LIN {X 0,Y 467.531,Z 199.445,A -85,B 0,C 180,E1 -7625.111,E2 -7625.111} C_VEL
LIN {X 0,Y 467.326,Z 207.202,A -85,B 0,C 180,E1 -7628.383,E2 -7628.383} C_VEL
LIN {X 0,Y 467.095,Z 214.915,A -85,B 0,C 180,E1 -7631.583,E2 -7631.583} C_VEL
LIN {X 0,Y 466.901,Z 222.309,A -85,B 0,C 180,E1 -7634.625,E2 -7634.625} C_VEL
LIN {X 0,Y 469.16,Z 236.323,A -85,B 0,C 180,E1 -7635.082,E2 -7635.082} C_VEL
LIN {X 0,Y 469.908,Z 243.542,A -85,B 0,C 180,E1 -7635.383,E2 -7635.383} C_VEL
LIN {X 0,Y 469.499,Z 254.745,A -85,B 0,C 180,E1 -7635.923,E2 -7635.923} C_VEL
LIN {X 0,Y 468.983,Z 266.744,A -85,B 0,C 180,E1 -7636.681,E2 -7636.681} C_VEL
LIN {X 0,Y 468.599,Z 277.34,A -85,B 0,C 180,E1 -7637.54,E2 -7637.54} C_VEL
LIN {X 0,Y 468.086,Z 287.224,A -85,B 0,C 180,E1 -7638.526,E2 -7638.526} C_VEL
LIN {X 0,Y 467.594,Z 296.115,A -85,B 0,C 180,E1 -7639.611,E2 -7639.611} C_VEL
LIN {X 0,Y 467.253,Z 304.795,A -85,B 0,C 180,E1 -7640.914,E2 -7640.914} C_VEL
LIN {X 0,Y 466.98,Z 311.72,A -85,B 0,C 180,E1 -7642.217,E2 -7642.217} C_VEL
LIN {X 0,Y 466.805,Z 317.387,A -85,B 0,C 180,E1 -7643.549,E2 -7643.549} C_VEL
LIN {X 0,Y 466.739,Z 321.625,A -85,B 0,C 180,E1 -7644.817,E2 -7644.817} C_VEL
LIN {X 0,Y 466.646,Z 323.927,A -85,B 0,C 180,E1 -7645.682,E2 -7645.682} C_VEL
LIN {X 0,Y 466.688,Z 325.799,A -85,B 0,C 180,E1 -7646.547,E2 -7646.547} C_VEL
LIN {X 0,Y 466.662,Z 327.203,A -85,B 0,C 180,E1 -7647.411,E2 -7647.411} C_VEL
LIN {X 0,Y 466.618,Z 328.815,A -85,B 0,C 180,E1 -7649.138,E2 -7649.138} C_VEL
LIN {X 0,Y 466.599,Z 329.038,A -85,B 0,C 180,E1 -7650.001,E2 -7650.001} C_VEL
LIN {X 0,Y 466.618,Z 328.829,A -85,B 0,C 180,E1 -7650.864,E2 -7650.864} C_VEL
LIN {X 0,Y 466.662,Z 327.238,A -85,B 0,C 180,E1 -7652.59,E2 -7652.59} C_VEL
LIN {X 0,Y 466.688,Z 325.85,A -85,B 0,C 180,E1 -7653.454,E2 -7653.454} C_VEL
LIN {X 0,Y 466.689,Z 322.925,A -85,B 0,C 180,E1 -7654.751,E2 -7654.751} C_VEL
LIN {X 0,Y 466.753,Z 318.967,A -85,B 0,C 180,E1 -7656.05,E2 -7656.05} C_VEL
LIN {X 0,Y 466.963,Z 312.888,A -85,B 0,C 180,E1 -7657.567,E2 -7657.567} C_VEL
LIN {X 0,Y 467.224,Z 306.239,A -85,B 0,C 180,E1 -7658.869,E2 -7658.869} C_VEL
LIN {X 0,Y 467.551,Z 297.991,A -85,B 0,C 180,E1 -7660.173,E2 -7660.173} C_VEL
LIN {X 0,Y 468.052,Z 289.556,A -85,B 0,C 180,E1 -7661.256,E2 -7661.256} C_VEL
LIN {X 0,Y 468.503,Z 279.581,A -85,B 0,C 180,E1 -7662.301,E2 -7662.301} C_VEL
LIN {X 0,Y 468.948,Z 268.843,A -85,B 0,C 180,E1 -7663.211,E2 -7663.211} C_VEL
LIN {X 0,Y 469.452,Z 257.578,A -85,B 0,C 180,E1 -7663.969,E2 -7663.969} C_VEL
LIN {X 0,Y 469.965,Z 246.132,A -85,B 0,C 180,E1 -7664.561,E2 -7664.561} C_VEL
LIN {X 0,Y 469.806,Z 241.144,A -85,B 0,C 180,E1 -7664.78,E2 -7664.78} C_VEL
LIN {X 0,Y 468.016,Z 228.536,A -85,B 0,C 180,E1 -7665.256,E2 -7665.256} C_VEL
LIN {X 0,Y 466.938,Z 222.233,A -85,B 0,C 180,E1 -7665.454,E2 -7665.454} C_VEL
LIN {X 0,Y 467.097,Z 214.666,A -85,B 0,C 180,E1 -7668.575,E2 -7668.575} C_VEL
LIN {X 0,Y 467.326,Z 207.444,A -85,B 0,C 180,E1 -7671.619,E2 -7671.619} C_VEL
LIN {X 0,Y 467.555,Z 199.754,A -85,B 0,C 180,E1 -7674.889,E2 -7674.889} C_VEL
LIN {X 0,Y 467.862,Z 192.074,A -85,B 0,C 180,E1 -7678.239,E2 -7678.239} C_VEL
LIN {X 0,Y 468.123,Z 186.635,A -85,B 0,C 180,E1 -7680.692,E2 -7680.692} C_VEL
LIN {X 0,Y 468.345,Z 182.022,A -85,B 0,C 180,E1 -7682.824,E2 -7682.824} C_VEL
LIN {X 0,Y 468.553,Z 176.91,A -85,B 0,C 180,E1 -7685.271,E2 -7685.271} C_VEL
LIN {X 0,Y 468.198,Z 172.916,A -85,B 0,C 180,E1 -7687.291,E2 -7687.291} C_VEL
LIN {X 0,Y 467.587,Z 169.247,A -85,B 0,C 180,E1 -7689.28,E2 -7689.28} C_VEL
LIN {X 0,Y 467.608,Z 169.237,A -85,B 0,C 180,E1 -7692.57,E2 -7692.57} C_VEL
LIN {X 0,Y 467.557,Z 169.245,A -85,B 0,C 180,E1 -7695.051,E2 -7695.051} C_VEL
LIN {X 0,Y 467.575,Z 169.243,A -85,B 0,C 180,E1 -7697.438,E2 -7697.438} C_VEL
LIN {X 0,Y 467.543,Z 169.247,A -85,B 0,C 180,E1 -7700.851,E2 -7700.851} C_VEL
LIN {X 0,Y 467.545,Z 169.243,A -85,B 0,C 180,E1 -7704.259,E2 -7704.259} C_VEL
LIN {X 0,Y 467.562,Z 169.245,A -85,B 0,C 180,E1 -7707.319,E2 -7707.319} C_VEL
LIN {X 0,Y 467.549,Z 169.247,A -85,B 0,C 180,E1 -7710.666,E2 -7710.666} C_VEL
LIN {X 0,Y 467.594,Z 169.241,A -85,B 0,C 180,E1 -7713.198,E2 -7713.198} C_VEL
LIN {X 0,Y 467.584,Z 169.24,A -85,B 0,C 180,E1 -7716.463,E2 -7716.463} C_VEL
LIN {X 0,Y 467.601,Z 169.237,A -85,B 0,C 180,E1 -7719.776,E2 -7719.776} C_VEL
LIN {X 0,Y 467.594,Z 169.242,A -85,B 0,C 180,E1 -7722.506,E2 -7722.506} C_VEL
LIN {X 0,Y 467.578,Z 169.243,A -85,B 0,C 180,E1 -7725.196,E2 -7725.196} C_VEL
LIN {X 0,Y 467.658,Z 169.231,A -85,B 0,C 180,E1 -7727.855,E2 -7727.855} C_VEL
LIN {X 0,Y 467.671,Z 169.227,A -85,B 0,C 180,E1 -7731.357,E2 -7731.357} C_VEL
LIN {X 0,Y 467.745,Z 169.222,A -85,B 0,C 180,E1 -7733.963,E2 -7733.963} C_VEL
LIN {X 0,Y 467.831,Z 169.21,A -85,B 0,C 180,E1 -7737.417,E2 -7737.417} C_VEL
LIN {X 0,Y 467.8,Z 169.213,A -85,B 0,C 180,E1 -7740.861,E2 -7740.861} C_VEL
LIN {X 0,Y 467.842,Z 169.208,A -85,B 0,C 180,E1 -7742.583,E2 -7742.583} C_VEL
LIN {X 0,Y 467.728,Z 169.225,A -85,B 0,C 180,E1 -7746.038,E2 -7746.038} C_VEL
LIN {X 0,Y 467.655,Z 169.232,A -85,B 0,C 180,E1 -7748.644,E2 -7748.644} C_VEL
LIN {X 0,Y 467.629,Z 169.238,A -85,B 0,C 180,E1 -7752.146,E2 -7752.146} C_VEL
LIN {X 0,Y 467.642,Z 169.235,A -85,B 0,C 180,E1 -7755.894,E2 -7755.894} C_VEL
LIN {X 0,Y 467.602,Z 169.241,A -85,B 0,C 180,E1 -7759.309,E2 -7759.309} C_VEL
LIN {X 0,Y 467.517,Z 169.25,A -85,B 0,C 180,E1 -7762.075,E2 -7762.075} C_VEL
LIN {X 0,Y 467.581,Z 169.241,A -85,B 0,C 180,E1 -7764.889,E2 -7764.889} C_VEL
LIN {X 0,Y 467.601,Z 169.239,A -85,B 0,C 180,E1 -7767.771,E2 -7767.771} C_VEL
LIN {X 0,Y 467.553,Z 169.248,A -85,B 0,C 180,E1 -7771.047,E2 -7771.047} C_VEL
LIN {X 0,Y 467.572,Z 169.242,A -85,B 0,C 180,E1 -7774.244,E2 -7774.244} C_VEL
LIN {X 0,Y 467.532,Z 169.249,A -85,B 0,C 180,E1 -7777.188,E2 -7777.188} C_VEL
LIN {X 0,Y 467.56,Z 169.242,A -85,B 0,C 180,E1 -7780.267,E2 -7780.267} C_VEL
LIN {X 0,Y 467.574,Z 169.243,A -85,B 0,C 180,E1 -7782.569,E2 -7782.569} C_VEL
LIN {X 0,Y 467.559,Z 169.244,A -85,B 0,C 180,E1 -7785.055,E2 -7785.055} C_VEL
LIN {X 0,Y 467.58,Z 169.241,A -85,B 0,C 180,E1 -7787.442,E2 -7787.442} C_VEL
LIN {X 0,Y 467.563,Z 169.244,A -85,B 0,C 180,E1 -7790.049,E2 -7790.049} C_VEL
LIN {X 0,Y 467.489,Z 169.254,A -85,B 0,C 180,E1 -7791.951,E2 -7791.951} C_VEL
LIN {X 0,Y 467.443,Z 170.109,A -85,B 0,C 180,E1 -7793.032,E2 -7793.032} C_VEL
LIN {X 0,Y 467.424,Z 173.846,A -85,B 0,C 180,E1 -7795.788,E2 -7795.788} C_VEL
LIN {X 0,Y 467.292,Z 178.365,A -85,B 0,C 180,E1 -7799.012,E2 -7799.012} C_VEL
LIN {X 0,Y 467.153,Z 182.951,A -85,B 0,C 180,E1 -7802.202,E2 -7802.202} C_VEL
LIN {X 0,Y 467.065,Z 187.177,A -85,B 0,C 180,E1 -7805.083,E2 -7805.083} C_VEL
LIN {X 0,Y 466.926,Z 191.458,A -85,B 0,C 180,E1 -7807.897,E2 -7807.897} C_VEL
LIN {X 0,Y 466.869,Z 196.787,A -85,B 0,C 180,E1 -7811.32,E2 -7811.32} C_VEL
LIN {X 0,Y 466.799,Z 198.848,A -85,B 0,C 180,E1 -7812.63,E2 -7812.63} C_VEL
LIN {X 0,Y 469.626,Z 212.179,A -85,B 0,C 180,E1 -7813.118,E2 -7813.118} C_VEL
LIN {X 0,Y 470.304,Z 216.846,A -85,B 0,C 180,E1 -7813.322,E2 -7813.322} C_VEL
LIN {X 0,Y 470.182,Z 221.204,A -85,B 0,C 180,E1 -7813.507,E2 -7813.507} C_VEL
LIN {X 0,Y 469.309,Z 226.817,A -85,B 0,C 180,E1 -7813.759,E2 -7813.759} C_VEL
LIN {X 0,Y 464.784,Z 238.986,A -85,B 0,C 180,E1 -7814.361,E2 -7814.361} C_VEL
LIN {X 0,Y 462.582,Z 245.641,A -85,B 0,C 180,E1 -7814.797,E2 -7814.797} C_VEL
LIN {X 0,Y 462.098,Z 248.855,A -85,B 0,C 180,E1 -7815.056,E2 -7815.056} C_VEL
LIN {X 0,Y 461.556,Z 259.922,A -85,B 0,C 180,E1 -7816.124,E2 -7816.124} C_VEL
LIN {X 0,Y 461.031,Z 269.785,A -85,B 0,C 180,E1 -7817.325,E2 -7817.325} C_VEL
LIN {X 0,Y 460.671,Z 278.005,A -85,B 0,C 180,E1 -7818.561,E2 -7818.561} C_VEL
LIN {X 0,Y 460.209,Z 285.169,A -85,B 0,C 180,E1 -7819.885,E2 -7819.885} C_VEL
LIN {X 0,Y 459.987,Z 290.869,A -85,B 0,C 180,E1 -7821.212,E2 -7821.212} C_VEL
LIN {X 0,Y 459.795,Z 295.352,A -85,B 0,C 180,E1 -7822.535,E2 -7822.535} C_VEL
LIN {X 0,Y 459.673,Z 298.757,A -85,B 0,C 180,E1 -7823.856,E2 -7823.856} C_VEL
LIN {X 0,Y 459.645,Z 300.447,A -85,B 0,C 180,E1 -7824.736,E2 -7824.736} C_VEL
LIN {X 0,Y 459.613,Z 302.633,A -85,B 0,C 180,E1 -7826.493,E2 -7826.493} C_VEL
LIN {X 0,Y 459.585,Z 303.127,A -85,B 0,C 180,E1 -7827.37,E2 -7827.37} C_VEL
LIN {X 0,Y 459.525,Z 302.9,A -85,B 0,C 180,E1 -7829.123,E2 -7829.123} C_VEL
LIN {X 0,Y 459.535,Z 302.217,A -85,B 0,C 180,E1 -7829.999,E2 -7829.999} C_VEL
LIN {X 0,Y 459.562,Z 301.135,A -85,B 0,C 180,E1 -7830.876,E2 -7830.876} C_VEL
LIN {X 0,Y 459.629,Z 299.611,A -85,B 0,C 180,E1 -7831.752,E2 -7831.752} C_VEL
LIN {X 0,Y 459.785,Z 296.553,A -85,B 0,C 180,E1 -7833.066,E2 -7833.066} C_VEL
LIN {X 0,Y 459.934,Z 292.454,A -85,B 0,C 180,E1 -7834.381,E2 -7834.381} C_VEL
LIN {X 0,Y 460.123,Z 286.196,A -85,B 0,C 180,E1 -7835.917,E2 -7835.917} C_VEL
LIN {X 0,Y 460.556,Z 278.996,A -85,B 0,C 180,E1 -7837.299,E2 -7837.299} C_VEL
LIN {X 0,Y 460.913,Z 270.853,A -85,B 0,C 180,E1 -7838.549,E2 -7838.549} C_VEL
LIN {X 0,Y 461.396,Z 262.105,A -85,B 0,C 180,E1 -7839.644,E2 -7839.644} C_VEL
LIN {X 0,Y 461.917,Z 251.339,A -85,B 0,C 180,E1 -7840.74,E2 -7840.74} C_VEL
LIN {X 0,Y 462.429,Z 240.492,A -85,B 0,C 180,E1 -7841.616,E2 -7841.616} C_VEL
LIN {X 0,Y 462.913,Z 228.195,A -85,B 0,C 180,E1 -7842.39,E2 -7842.39} C_VEL
LIN {X 0,Y 463.294,Z 216.584,A -85,B 0,C 180,E1 -7842.94,E2 -7842.94} C_VEL
LIN {X 0,Y 460.702,Z 203.549,A -85,B 0,C 180,E1 -7843.468,E2 -7843.468} C_VEL
LIN {X 0,Y 459.742,Z 199.024,A -85,B 0,C 180,E1 -7843.611,E2 -7843.611} C_VEL
LIN {X 0,Y 459.855,Z 195.331,A -85,B 0,C 180,E1 -7845.966,E2 -7845.966} C_VEL
LIN {X 0,Y 459.885,Z 191.089,A -85,B 0,C 180,E1 -7848.717,E2 -7848.717} C_VEL
LIN {X 0,Y 460.003,Z 186.877,A -85,B 0,C 180,E1 -7851.508,E2 -7851.508} C_VEL
LIN {X 0,Y 460.086,Z 182.722,A -85,B 0,C 180,E1 -7854.355,E2 -7854.355} C_VEL
LIN {X 0,Y 460.199,Z 177.984,A -85,B 0,C 180,E1 -7857.654,E2 -7857.654} C_VEL
LIN {X 0,Y 460.313,Z 174.331,A -85,B 0,C 180,E1 -7860.251,E2 -7860.251} C_VEL
LIN {X 0,Y 460.352,Z 170.15,A -85,B 0,C 180,E1 -7863.336,E2 -7863.336} C_VEL
LIN {X 0,Y 460.481,Z 170.125,A -85,B 0,C 180,E1 -7866.01,E2 -7866.01} C_VEL
LIN {X 0,Y 460.52,Z 170.123,A -85,B 0,C 180,E1 -7868.893,E2 -7868.893} C_VEL
LIN {X 0,Y 460.509,Z 170.122,A -85,B 0,C 180,E1 -7872.178,E2 -7872.178} C_VEL
LIN {X 0,Y 460.504,Z 170.125,A -85,B 0,C 180,E1 -7875.409,E2 -7875.409} C_VEL
LIN {X 0,Y 460.526,Z 170.117,A -85,B 0,C 180,E1 -7878.393,E2 -7878.393} C_VEL
LIN {X 0,Y 460.521,Z 170.12,A -85,B 0,C 180,E1 -7881.266,E2 -7881.266} C_VEL
LIN {X 0,Y 460.486,Z 170.127,A -85,B 0,C 180,E1 -7884.552,E2 -7884.552} C_VEL
LIN {X 0,Y 460.506,Z 170.122,A -85,B 0,C 180,E1 -7887.713,E2 -7887.713} C_VEL
LIN {X 0,Y 460.52,Z 170.122,A -85,B 0,C 180,E1 -7890.767,E2 -7890.767} C_VEL
LIN {X 0,Y 460.543,Z 170.115,A -85,B 0,C 180,E1 -7893.733,E2 -7893.733} C_VEL
LIN {X 0,Y 460.531,Z 170.121,A -85,B 0,C 180,E1 -7896.623,E2 -7896.623} C_VEL
LIN {X 0,Y 460.54,Z 170.117,A -85,B 0,C 180,E1 -7899.452,E2 -7899.452} C_VEL
LIN {X 0,Y 460.526,Z 170.121,A -85,B 0,C 180,E1 -7902.228,E2 -7902.228} C_VEL
LIN {X 0,Y 460.54,Z 170.119,A -85,B 0,C 180,E1 -7904.964,E2 -7904.964} C_VEL
LIN {X 0,Y 460.642,Z 170.105,A -85,B 0,C 180,E1 -7907.666,E2 -7907.666} C_VEL
LIN {X 0,Y 460.635,Z 170.104,A -85,B 0,C 180,E1 -7911.224,E2 -7911.224} C_VEL
LIN {X 0,Y 460.701,Z 170.102,A -85,B 0,C 180,E1 -7913.87,E2 -7913.87} C_VEL
LIN {X 0,Y 460.789,Z 170.089,A -85,B 0,C 180,E1 -7917.377,E2 -7917.377} C_VEL
LIN {X 0,Y 460.812,Z 170.084,A -85,B 0,C 180,E1 -7920,E2 -7920} C_VEL
LIN {X 0,Y 460.798,Z 170.086,A -85,B 0,C 180,E1 -7922.622,E2 -7922.622} C_VEL
LIN {X 0,Y 460.693,Z 170.099,A -85,B 0,C 180,E1 -7926.13,E2 -7926.13} C_VEL
LIN {X 0,Y 460.634,Z 170.104,A -85,B 0,C 180,E1 -7928.776,E2 -7928.776} C_VEL
LIN {X 0,Y 460.616,Z 170.107,A -85,B 0,C 180,E1 -7932.467,E2 -7932.467} C_VEL
LIN {X 0,Y 460.566,Z 170.115,A -85,B 0,C 180,E1 -7935.999,E2 -7935.999} C_VEL
LIN {X 0,Y 460.536,Z 170.119,A -85,B 0,C 180,E1 -7938.903,E2 -7938.903} C_VEL
LIN {X 0,Y 460.532,Z 170.121,A -85,B 0,C 180,E1 -7941.485,E2 -7941.485} C_VEL
LIN {X 0,Y 460.528,Z 170.118,A -85,B 0,C 180,E1 -7944.333,E2 -7944.333} C_VEL
LIN {X 0,Y 460.554,Z 170.116,A -85,B 0,C 180,E1 -7947.245,E2 -7947.245} C_VEL
LIN {X 0,Y 460.498,Z 170.123,A -85,B 0,C 180,E1 -7950.241,E2 -7950.241} C_VEL
LIN {X 0,Y 460.502,Z 170.123,A -85,B 0,C 180,E1 -7953.327,E2 -7953.327} C_VEL
LIN {X 0,Y 460.453,Z 170.129,A -85,B 0,C 180,E1 -7956.532,E2 -7956.532} C_VEL
LIN {X 0,Y 460.555,Z 170.116,A -85,B 0,C 180,E1 -7959.86,E2 -7959.86} C_VEL
LIN {X 0,Y 460.521,Z 170.12,A -85,B 0,C 180,E1 -7962.907,E2 -7962.907} C_VEL
LIN {X 0,Y 460.505,Z 170.125,A -85,B 0,C 180,E1 -7965.831,E2 -7965.831} C_VEL
LIN {X 0,Y 460.517,Z 170.126,A -85,B 0,C 180,E1 -7968.992,E2 -7968.992} C_VEL
LIN {X 0,Y 460.582,Z 170.329,A -85,B 0,C 180,E1 -7971.097,E2 -7971.097} C_VEL
LIN {X 0,Y 461.37,Z 175.587,A -85,B 0,C 180,E1 -7973.837,E2 -7973.837} C_VEL
LIN {X 0,Y 461.328,Z 180.521,A -85,B 0,C 180,E1 -7976.22,E2 -7976.22} C_VEL
LIN {X 0,Y 461.027,Z 188.217,A -85,B 0,C 180,E1 -7979.801,E2 -7979.801} C_VEL
LIN {X 0,Y 460.628,Z 195.961,A -85,B 0,C 180,E1 -7983.253,E2 -7983.253} C_VEL
LIN {X 0,Y 460.341,Z 203.089,A -85,B 0,C 180,E1 -7986.351,E2 -7986.351} C_VEL
LIN {X 0,Y 460.235,Z 208.512,A -85,B 0,C 180,E1 -7988.67,E2 -7988.67} C_VEL
LIN {X 0,Y 459.991,Z 215.835,A -85,B 0,C 180,E1 -7991.756,E2 -7991.756} C_VEL
LIN {X 0,Y 459.837,Z 222.228,A -85,B 0,C 180,E1 -7994.405,E2 -7994.405} C_VEL
LIN {X 0,Y 461.957,Z 235.144,A -85,B 0,C 180,E1 -7994.818,E2 -7994.818} C_VEL
LIN {X 0,Y 462.974,Z 244.425,A -85,B 0,C 180,E1 -7995.215,E2 -7995.215} C_VEL
LIN {X 0,Y 462.509,Z 256.356,A -85,B 0,C 180,E1 -7995.818,E2 -7995.818} C_VEL
LIN {X 0,Y 461.959,Z 267.864,A -85,B 0,C 180,E1 -7996.586,E2 -7996.586} C_VEL
LIN {X 0,Y 461.5,Z 279.085,A -85,B 0,C 180,E1 -7997.539,E2 -7997.539} C_VEL
LIN {X 0,Y 460.984,Z 288.904,A -85,B 0,C 180,E1 -7998.57,E2 -7998.57} C_VEL
LIN {X 0,Y 460.498,Z 297.458,A -85,B 0,C 180,E1 -7999.671,E2 -7999.671} C_VEL
LIN {X 0,Y 460.14,Z 305.785,A -85,B 0,C 180,E1 -8000.994,E2 -8000.994} C_VEL
LIN {X 0,Y 459.879,Z 312.496,A -85,B 0,C 180,E1 -8002.317,E2 -8002.317} C_VEL
LIN {X 0,Y 459.668,Z 318.645,A -85,B 0,C 180,E1 -8003.857,E2 -8003.857} C_VEL
LIN {X 0,Y 459.617,Z 322.637,A -85,B 0,C 180,E1 -8005.177,E2 -8005.177} C_VEL
LIN {X 0,Y 459.583,Z 325.586,A -85,B 0,C 180,E1 -8006.494,E2 -8006.494} C_VEL
LIN {X 0,Y 459.584,Z 326.995,A -85,B 0,C 180,E1 -8007.371,E2 -8007.371} C_VEL
LIN {X 0,Y 459.521,Z 328.613,A -85,B 0,C 180,E1 -8009.124,E2 -8009.124} C_VEL
LIN {X 0,Y 459.531,Z 328.84,A -85,B 0,C 180,E1 -8010.001,E2 -8010.001} C_VEL
LIN {X 0,Y 459.521,Z 328.636,A -85,B 0,C 180,E1 -8010.877,E2 -8010.877} C_VEL
LIN {X 0,Y 459.584,Z 327.051,A -85,B 0,C 180,E1 -8012.63,E2 -8012.63} C_VEL
LIN {X 0,Y 459.583,Z 325.667,A -85,B 0,C 180,E1 -8013.507,E2 -8013.507} C_VEL
LIN {X 0,Y 459.616,Z 322.747,A -85,B 0,C 180,E1 -8014.825,E2 -8014.825} C_VEL
LIN {X 0,Y 459.714,Z 317.778,A -85,B 0,C 180,E1 -8016.431,E2 -8016.431} C_VEL
LIN {X 0,Y 459.923,Z 311.717,A -85,B 0,C 180,E1 -8017.905,E2 -8017.905} C_VEL
LIN {X 0,Y 460.227,Z 304.854,A -85,B 0,C 180,E1 -8019.227,E2 -8019.227} C_VEL
LIN {X 0,Y 460.535,Z 297.853,A -85,B 0,C 180,E1 -8020.329,E2 -8020.329} C_VEL
LIN {X 0,Y 461.076,Z 289.433,A -85,B 0,C 180,E1 -8021.429,E2 -8021.429} C_VEL
LIN {X 0,Y 461.531,Z 279.689,A -85,B 0,C 180,E1 -8022.47,E2 -8022.47} C_VEL
LIN {X 0,Y 462.036,Z 268.766,A -85,B 0,C 180,E1 -8023.412,E2 -8023.412} C_VEL
LIN {X 0,Y 462.578,Z 257.531,A -85,B 0,C 180,E1 -8024.181,E2 -8024.181} C_VEL
LIN {X 0,Y 463.098,Z 246.138,A -85,B 0,C 180,E1 -8024.782,E2 -8024.782} C_VEL
LIN {X 0,Y 462.767,Z 240.436,A -85,B 0,C 180,E1 -8025.041,E2 -8025.041} C_VEL
LIN {X 0,Y 460.923,Z 228.115,A -85,B 0,C 180,E1 -8025.512,E2 -8025.512} C_VEL
LIN {X 0,Y 459.867,Z 222.077,A -85,B 0,C 180,E1 -8025.693,E2 -8025.693} C_VEL
LIN {X 0,Y 460.061,Z 213.819,A -85,B 0,C 180,E1 -8029.173,E2 -8029.173} C_VEL
LIN {X 0,Y 460.298,Z 206.234,A -85,B 0,C 180,E1 -8032.439,E2 -8032.439} C_VEL
LIN {X 0,Y 460.581,Z 198.482,A -85,B 0,C 180,E1 -8035.805,E2 -8035.805} C_VEL
LIN {X 0,Y 460.948,Z 190.901,A -85,B 0,C 180,E1 -8039.201,E2 -8039.201} C_VEL
LIN {X 0,Y 461.257,Z 184.397,A -85,B 0,C 180,E1 -8042.226,E2 -8042.226} C_VEL
LIN {X 0,Y 461.513,Z 179.286,A -85,B 0,C 180,E1 -8044.682,E2 -8044.682} C_VEL
LIN {X 0,Y 461.282,Z 174.713,A -85,B 0,C 180,E1 -8046.997,E2 -8046.997} C_VEL
LIN {X 0,Y 460.551,Z 170.124,A -85,B 0,C 180,E1 -8049.48,E2 -8049.48} C_VEL
LIN {X 0,Y 460.531,Z 170.118,A -85,B 0,C 180,E1 -8052.903,E2 -8052.903} C_VEL
LIN {X 0,Y 460.497,Z 170.124,A -85,B 0,C 180,E1 -8055.829,E2 -8055.829} C_VEL
LIN {X 0,Y 460.514,Z 170.123,A -85,B 0,C 180,E1 -8058.987,E2 -8058.987} C_VEL
LIN {X 0,Y 460.501,Z 170.123,A -85,B 0,C 180,E1 -8061.264,E2 -8061.264} C_VEL
LIN {X 0,Y 460.495,Z 170.121,A -85,B 0,C 180,E1 -8064.553,E2 -8064.553} C_VEL
LIN {X 0,Y 460.512,Z 170.121,A -85,B 0,C 180,E1 -8067.714,E2 -8067.714} C_VEL
LIN {X 0,Y 460.519,Z 170.123,A -85,B 0,C 180,E1 -8070.768,E2 -8070.768} C_VEL
LIN {X 0,Y 460.54,Z 170.118,A -85,B 0,C 180,E1 -8073.733,E2 -8073.733} C_VEL
LIN {X 0,Y 460.537,Z 170.118,A -85,B 0,C 180,E1 -8076.624,E2 -8076.624} C_VEL
LIN {X 0,Y 460.548,Z 170.116,A -85,B 0,C 180,E1 -8079.453,E2 -8079.453} C_VEL
LIN {X 0,Y 460.544,Z 170.118,A -85,B 0,C 180,E1 -8082.23,E2 -8082.23} C_VEL
LIN {X 0,Y 460.541,Z 170.119,A -85,B 0,C 180,E1 -8084.964,E2 -8084.964} C_VEL
LIN {X 0,Y 460.604,Z 170.109,A -85,B 0,C 180,E1 -8087.666,E2 -8087.666} C_VEL
LIN {X 0,Y 460.616,Z 170.106,A -85,B 0,C 180,E1 -8091.224,E2 -8091.224} C_VEL
LIN {X 0,Y 460.709,Z 170.097,A -85,B 0,C 180,E1 -8093.87,E2 -8093.87} C_VEL
LIN {X 0,Y 460.772,Z 170.089,A -85,B 0,C 180,E1 -8097.378,E2 -8097.378} C_VEL
LIN {X 0,Y 460.82,Z 170.084,A -85,B 0,C 180,E1 -8100,E2 -8100} C_VEL
LIN {X 0,Y 460.807,Z 170.084,A -85,B 0,C 180,E1 -8102.623,E2 -8102.623} C_VEL
LIN {X 0,Y 460.692,Z 170.1,A -85,B 0,C 180,E1 -8106.13,E2 -8106.13} C_VEL
LIN {X 0,Y 460.602,Z 170.11,A -85,B 0,C 180,E1 -8108.777,E2 -8108.777} C_VEL
LIN {X 0,Y 460.582,Z 170.114,A -85,B 0,C 180,E1 -8112.335,E2 -8112.335} C_VEL
LIN {X 0,Y 460.598,Z 170.111,A -85,B 0,C 180,E1 -8116.008,E2 -8116.008} C_VEL
LIN {X 0,Y 460.552,Z 170.116,A -85,B 0,C 180,E1 -8118.905,E2 -8118.905} C_VEL
LIN {X 0,Y 460.494,Z 170.125,A -85,B 0,C 180,E1 -8121.487,E2 -8121.487} C_VEL
LIN {X 0,Y 460.52,Z 170.12,A -85,B 0,C 180,E1 -8124.334,E2 -8124.334} C_VEL
LIN {X 0,Y 460.552,Z 170.118,A -85,B 0,C 180,E1 -8127.246,E2 -8127.246} C_VEL
LIN {X 0,Y 460.507,Z 170.12,A -85,B 0,C 180,E1 -8130.241,E2 -8130.241} C_VEL
LIN {X 0,Y 460.512,Z 170.122,A -85,B 0,C 180,E1 -8133.327,E2 -8133.327} C_VEL
LIN {X 0,Y 460.461,Z 170.129,A -85,B 0,C 180,E1 -8136.531,E2 -8136.531} C_VEL
LIN {X 0,Y 460.512,Z 170.12,A -85,B 0,C 180,E1 -8139.865,E2 -8139.865} C_VEL
LIN {X 0,Y 460.501,Z 170.125,A -85,B 0,C 180,E1 -8142.902,E2 -8142.902} C_VEL
LIN {X 0,Y 460.499,Z 170.122,A -85,B 0,C 180,E1 -8145.833,E2 -8145.833} C_VEL
LIN {X 0,Y 460.521,Z 170.122,A -85,B 0,C 180,E1 -8148.991,E2 -8148.991} C_VEL
LIN {X 0,Y 460.487,Z 170.129,A -85,B 0,C 180,E1 -8151.266,E2 -8151.266} C_VEL
LIN {X 0,Y 460.417,Z 170.38,A -85,B 0,C 180,E1 -8152.538,E2 -8152.538} C_VEL
LIN {X 0,Y 460.384,Z 174.49,A -85,B 0,C 180,E1 -8155.612,E2 -8155.612} C_VEL
LIN {X 0,Y 460.247,Z 178.859,A -85,B 0,C 180,E1 -8158.774,E2 -8158.774} C_VEL
LIN {X 0,Y 460.13,Z 183.054,A -85,B 0,C 180,E1 -8161.74,E2 -8161.74} C_VEL
LIN {X 0,Y 460.031,Z 187.293,A -85,B 0,C 180,E1 -8164.676,E2 -8164.676} C_VEL
LIN {X 0,Y 459.894,Z 191.585,A -85,B 0,C 180,E1 -8167.541,E2 -8167.541} C_VEL
LIN {X 0,Y 459.81,Z 195.898,A -85,B 0,C 180,E1 -8170.352,E2 -8170.352} C_VEL
LIN {X 0,Y 459.777,Z 199.096,A -85,B 0,C 180,E1 -8172.381,E2 -8172.381} C_VEL
LIN {X 0,Y 462.572,Z 212.162,A -85,B 0,C 180,E1 -8172.867,E2 -8172.867} C_VEL
LIN {X 0,Y 463.429,Z 218.062,A -85,B 0,C 180,E1 -8173.133,E2 -8173.133} C_VEL
LIN {X 0,Y 463.017,Z 230.357,A -85,B 0,C 180,E1 -8173.742,E2 -8173.742} C_VEL
LIN {X 0,Y 462.494,Z 241.477,A -85,B 0,C 180,E1 -8174.466,E2 -8174.466} C_VEL
LIN {X 0,Y 462.098,Z 248.855,A -85,B 0,C 180,E1 -8175.056,E2 -8175.056} C_VEL
LIN {X 0,Y 461.185,Z 253.695,A -85,B 0,C 180,E1 -8175.47,E2 -8175.47} C_VEL
LIN {X 0,Y 457.983,Z 261.265,A -85,B 0,C 180,E1 -8176.168,E2 -8176.168} C_VEL
LIN {X 0,Y 454.793,Z 268.356,A -85,B 0,C 180,E1 -8176.944,E2 -8176.944} C_VEL
LIN {X 0,Y 453.894,Z 272.311,A -85,B 0,C 180,E1 -8177.473,E2 -8177.473} C_VEL
LIN {X 0,Y 453.547,Z 280.639,A -85,B 0,C 180,E1 -8178.832,E2 -8178.832} C_VEL
LIN {X 0,Y 453.126,Z 287.296,A -85,B 0,C 180,E1 -8180.177,E2 -8180.177} C_VEL
LIN {X 0,Y 452.875,Z 292.598,A -85,B 0,C 180,E1 -8181.522,E2 -8181.522} C_VEL
LIN {X 0,Y 452.669,Z 296.728,A -85,B 0,C 180,E1 -8182.865,E2 -8182.865} C_VEL
LIN {X 0,Y 452.607,Z 298.91,A -85,B 0,C 180,E1 -8183.76,E2 -8183.76} C_VEL
LIN {X 0,Y 452.558,Z 300.61,A -85,B 0,C 180,E1 -8184.653,E2 -8184.653} C_VEL
LIN {X 0,Y 452.51,Z 302.812,A -85,B 0,C 180,E1 -8186.438,E2 -8186.438} C_VEL
LIN {X 0,Y 452.51,Z 303.319,A -85,B 0,C 180,E1 -8187.329,E2 -8187.329} C_VEL
LIN {X 0,Y 452.432,Z 303.109,A -85,B 0,C 180,E1 -8189.109,E2 -8189.109} C_VEL
LIN {X 0,Y 452.468,Z 301.365,A -85,B 0,C 180,E1 -8190.889,E2 -8190.889} C_VEL
LIN {X 0,Y 452.54,Z 299.85,A -85,B 0,C 180,E1 -8191.779,E2 -8191.779} C_VEL
LIN {X 0,Y 452.707,Z 296.809,A -85,B 0,C 180,E1 -8193.114,E2 -8193.114} C_VEL
LIN {X 0,Y 452.858,Z 292.728,A -85,B 0,C 180,E1 -8194.449,E2 -8194.449} C_VEL
LIN {X 0,Y 453.082,Z 286.487,A -85,B 0,C 180,E1 -8196.009,E2 -8196.009} C_VEL
LIN {X 0,Y 453.494,Z 279.813,A -85,B 0,C 180,E1 -8197.322,E2 -8197.322} C_VEL
LIN {X 0,Y 453.8,Z 272.756,A -85,B 0,C 180,E1 -8198.459,E2 -8198.459} C_VEL
LIN {X 0,Y 454.329,Z 264.4,A -85,B 0,C 180,E1 -8199.571,E2 -8199.571} C_VEL
LIN {X 0,Y 454.903,Z 254.082,A -85,B 0,C 180,E1 -8200.683,E2 -8200.683} C_VEL
LIN {X 0,Y 455.281,Z 243.881,A -85,B 0,C 180,E1 -8201.575,E2 -8201.575} C_VEL
LIN {X 0,Y 455.85,Z 232.71,A -85,B 0,C 180,E1 -8202.35,E2 -8202.35} C_VEL
LIN {X 0,Y 456.351,Z 221.033,A -85,B 0,C 180,E1 -8202.975,E2 -8202.975} C_VEL
LIN {X 0,Y 456.367,Z 217.337,A -85,B 0,C 180,E1 -8203.137,E2 -8203.137} C_VEL
LIN {X 0,Y 453.812,Z 204.467,A -85,B 0,C 180,E1 -8203.679,E2 -8203.679} C_VEL
LIN {X 0,Y 452.675,Z 199.183,A -85,B 0,C 180,E1 -8203.865,E2 -8203.865} C_VEL
LIN {X 0,Y 452.788,Z 195.543,A -85,B 0,C 180,E1 -8206.222,E2 -8206.222} C_VEL
LIN {X 0,Y 452.812,Z 191.277,A -85,B 0,C 180,E1 -8209.02,E2 -8209.02} C_VEL
LIN {X 0,Y 452.94,Z 187.055,A -85,B 0,C 180,E1 -8211.861,E2 -8211.861} C_VEL
LIN {X 0,Y 453.027,Z 182.89,A -85,B 0,C 180,E1 -8214.76,E2 -8214.76} C_VEL
LIN {X 0,Y 453.161,Z 178.496,A -85,B 0,C 180,E1 -8217.87,E2 -8217.87} C_VEL
LIN {X 0,Y 453.288,Z 174.467,A -85,B 0,C 180,E1 -8220.77,E2 -8220.77} C_VEL
LIN {X 0,Y 453.334,Z 171.255,A -85,B 0,C 180,E1 -8223.158,E2 -8223.158} C_VEL
LIN {X 0,Y 453.42,Z 171.007,A -85,B 0,C 180,E1 -8224.991,E2 -8224.991} C_VEL
LIN {X 0,Y 453.446,Z 171.002,A -85,B 0,C 180,E1 -8228.309,E2 -8228.309} C_VEL
LIN {X 0,Y 453.48,Z 170.998,A -85,B 0,C 180,E1 -8230.606,E2 -8230.606} C_VEL
LIN {X 0,Y 453.447,Z 171.003,A -85,B 0,C 180,E1 -8233.242,E2 -8233.242} C_VEL
LIN {X 0,Y 453.459,Z 170.999,A -85,B 0,C 180,E1 -8235.777,E2 -8235.777} C_VEL
LIN {X 0,Y 453.477,Z 170.995,A -85,B 0,C 180,E1 -8238.208,E2 -8238.208} C_VEL
LIN {X 0,Y 453.508,Z 170.997,A -85,B 0,C 180,E1 -8240.785,E2 -8240.785} C_VEL
LIN {X 0,Y 453.43,Z 171.003,A -85,B 0,C 180,E1 -8243.914,E2 -8243.914} C_VEL
LIN {X 0,Y 453.457,Z 171.002,A -85,B 0,C 180,E1 -8247.149,E2 -8247.149} C_VEL
LIN {X 0,Y 453.488,Z 170.996,A -85,B 0,C 180,E1 -8250.269,E2 -8250.269} C_VEL
LIN {X 0,Y 453.487,Z 170.995,A -85,B 0,C 180,E1 -8253.292,E2 -8253.292} C_VEL
LIN {X 0,Y 453.49,Z 170.997,A -85,B 0,C 180,E1 -8256.238,E2 -8256.238} C_VEL
LIN {X 0,Y 453.486,Z 170.996,A -85,B 0,C 180,E1 -8259.117,E2 -8259.117} C_VEL
LIN {X 0,Y 453.478,Z 171,A -85,B 0,C 180,E1 -8261.943,E2 -8261.943} C_VEL
LIN {X 0,Y 453.519,Z 170.995,A -85,B 0,C 180,E1 -8264.725,E2 -8264.725} C_VEL
LIN {X 0,Y 453.568,Z 170.987,A -85,B 0,C 180,E1 -8267.471,E2 -8267.471} C_VEL
LIN {X 0,Y 453.589,Z 170.981,A -85,B 0,C 180,E1 -8271.086,E2 -8271.086} C_VEL
LIN {X 0,Y 453.666,Z 170.976,A -85,B 0,C 180,E1 -8273.774,E2 -8273.774} C_VEL
LIN {X 0,Y 453.73,Z 170.967,A -85,B 0,C 180,E1 -8277.336,E2 -8277.336} C_VEL
LIN {X 0,Y 453.783,Z 170.96,A -85,B 0,C 180,E1 -8280,E2 -8280} C_VEL
LIN {X 0,Y 453.739,Z 170.965,A -85,B 0,C 180,E1 -8282.663,E2 -8282.663} C_VEL
LIN {X 0,Y 453.658,Z 170.975,A -85,B 0,C 180,E1 -8286.225,E2 -8286.225} C_VEL
LIN {X 0,Y 453.587,Z 170.982,A -85,B 0,C 180,E1 -8288.913,E2 -8288.913} C_VEL
LIN {X 0,Y 453.567,Z 170.985,A -85,B 0,C 180,E1 -8292.552,E2 -8292.552} C_VEL
LIN {X 0,Y 453.51,Z 170.993,A -85,B 0,C 180,E1 -8296.197,E2 -8296.197} C_VEL
LIN {X 0,Y 453.486,Z 170.997,A -85,B 0,C 180,E1 -8299.042,E2 -8299.042} C_VEL
LIN {X 0,Y 453.473,Z 170.998,A -85,B 0,C 180,E1 -8301.836,E2 -8301.836} C_VEL
LIN {X 0,Y 453.502,Z 170.995,A -85,B 0,C 180,E1 -8304.735,E2 -8304.735} C_VEL
LIN {X 0,Y 453.509,Z 170.991,A -85,B 0,C 180,E1 -8307.963,E2 -8307.963} C_VEL
LIN {X 0,Y 453.455,Z 171.002,A -85,B 0,C 180,E1 -8310.761,E2 -8310.761} C_VEL
LIN {X 0,Y 453.45,Z 171.001,A -85,B 0,C 180,E1 -8313.915,E2 -8313.915} C_VEL
LIN {X 0,Y 453.446,Z 171.003,A -85,B 0,C 180,E1 -8317.19,E2 -8317.19} C_VEL
LIN {X 0,Y 453.51,Z 170.993,A -85,B 0,C 180,E1 -8319.448,E2 -8319.448} C_VEL
LIN {X 0,Y 453.471,Z 170.997,A -85,B 0,C 180,E1 -8322.994,E2 -8322.994} C_VEL
LIN {X 0,Y 453.458,Z 171.002,A -85,B 0,C 180,E1 -8325.783,E2 -8325.783} C_VEL
LIN {X 0,Y 453.468,Z 171.005,A -85,B 0,C 180,E1 -8328.213,E2 -8328.213} C_VEL
LIN {X 0,Y 453.524,Z 171.014,A -85,B 0,C 180,E1 -8330.789,E2 -8330.789} C_VEL
LIN {X 0,Y 454.399,Z 177.085,A -85,B 0,C 180,E1 -8334.008,E2 -8334.008} C_VEL
LIN {X 0,Y 454.328,Z 181.48,A -85,B 0,C 180,E1 -8336.163,E2 -8336.163} C_VEL
LIN {X 0,Y 454.02,Z 188.076,A -85,B 0,C 180,E1 -8339.284,E2 -8339.284} C_VEL
LIN {X 0,Y 453.633,Z 194.696,A -85,B 0,C 180,E1 -8342.307,E2 -8342.307} C_VEL
LIN {X 0,Y 453.419,Z 201.324,A -85,B 0,C 180,E1 -8345.263,E2 -8345.263} C_VEL
LIN {X 0,Y 453.189,Z 208.757,A -85,B 0,C 180,E1 -8348.509,E2 -8348.509} C_VEL
LIN {X 0,Y 452.906,Z 216.714,A -85,B 0,C 180,E1 -8351.922,E2 -8351.922} C_VEL
LIN {X 0,Y 452.77,Z 221.945,A -85,B 0,C 180,E1 -8354.161,E2 -8354.161} C_VEL
LIN {X 0,Y 454.95,Z 235.448,A -85,B 0,C 180,E1 -8354.608,E2 -8354.608} C_VEL
LIN {X 0,Y 456.076,Z 245.296,A -85,B 0,C 180,E1 -8355.044,E2 -8355.044} C_VEL
LIN {X 0,Y 455.523,Z 257.787,A -85,B 0,C 180,E1 -8355.71,E2 -8355.71} C_VEL
LIN {X 0,Y 454.948,Z 268.969,A -85,B 0,C 180,E1 -8356.49,E2 -8356.49} C_VEL
LIN {X 0,Y 454.524,Z 279.015,A -85,B 0,C 180,E1 -8357.367,E2 -8357.367} C_VEL
LIN {X 0,Y 453.986,Z 288.62,A -85,B 0,C 180,E1 -8358.391,E2 -8358.391} C_VEL
LIN {X 0,Y 453.479,Z 297.194,A -85,B 0,C 180,E1 -8359.509,E2 -8359.509} C_VEL
LIN {X 0,Y 453.1,Z 305.534,A -85,B 0,C 180,E1 -8360.853,E2 -8360.853} C_VEL
LIN {X 0,Y 452.809,Z 312.255,A -85,B 0,C 180,E1 -8362.196,E2 -8362.196} C_VEL
LIN {X 0,Y 452.602,Z 318.416,A -85,B 0,C 180,E1 -8363.761,E2 -8363.761} C_VEL
LIN {X 0,Y 452.546,Z 322.417,A -85,B 0,C 180,E1 -8365.101,E2 -8365.101} C_VEL
LIN {X 0,Y 452.48,Z 325.37,A -85,B 0,C 180,E1 -8366.439,E2 -8366.439} C_VEL
LIN {X 0,Y 452.507,Z 326.786,A -85,B 0,C 180,E1 -8367.33,E2 -8367.33} C_VEL
LIN {X 0,Y 452.428,Z 328.41,A -85,B 0,C 180,E1 -8369.111,E2 -8369.111} C_VEL
LIN {X 0,Y 452.435,Z 328.642,A -85,B 0,C 180,E1 -8370.001,E2 -8370.001} C_VEL
LIN {X 0,Y 452.428,Z 328.443,A -85,B 0,C 180,E1 -8370.891,E2 -8370.891} C_VEL
LIN {X 0,Y 452.508,Z 326.865,A -85,B 0,C 180,E1 -8372.671,E2 -8372.671} C_VEL
LIN {X 0,Y 452.479,Z 325.484,A -85,B 0,C 180,E1 -8373.562,E2 -8373.562} C_VEL
LIN {X 0,Y 452.545,Z 322.571,A -85,B 0,C 180,E1 -8374.9,E2 -8374.9} C_VEL
LIN {X 0,Y 452.61,Z 318.106,A -85,B 0,C 180,E1 -8376.396,E2 -8376.396} C_VEL
LIN {X 0,Y 452.806,Z 313.556,A -85,B 0,C 180,E1 -8377.581,E2 -8377.581} C_VEL
LIN {X 0,Y 453.085,Z 307.179,A -85,B 0,C 180,E1 -8378.923,E2 -8378.923} C_VEL
LIN {X 0,Y 453.449,Z 299.208,A -85,B 0,C 180,E1 -8380.267,E2 -8380.267} C_VEL
LIN {X 0,Y 453.974,Z 291.099,A -85,B 0,C 180,E1 -8381.384,E2 -8381.384} C_VEL
LIN {X 0,Y 454.522,Z 281.213,A -85,B 0,C 180,E1 -8382.502,E2 -8382.502} C_VEL
LIN {X 0,Y 454.967,Z 271.506,A -85,B 0,C 180,E1 -8383.397,E2 -8383.397} C_VEL
LIN {X 0,Y 455.514,Z 261.023,A -85,B 0,C 180,E1 -8384.177,E2 -8384.177} C_VEL
LIN {X 0,Y 456.158,Z 248.407,A -85,B 0,C 180,E1 -8384.898,E2 -8384.898} C_VEL
LIN {X 0,Y 456.013,Z 242.327,A -85,B 0,C 180,E1 -8385.188,E2 -8385.188} C_VEL
LIN {X 0,Y 454.172,Z 229.559,A -85,B 0,C 180,E1 -8385.715,E2 -8385.715} C_VEL
LIN {X 0,Y 452.764,Z 221.88,A -85,B 0,C 180,E1 -8385.958,E2 -8385.958} C_VEL
LIN {X 0,Y 452.974,Z 214.779,A -85,B 0,C 180,E1 -8389.014,E2 -8389.014} C_VEL
LIN {X 0,Y 453.244,Z 207.188,A -85,B 0,C 180,E1 -8392.326,E2 -8392.326} C_VEL
LIN {X 0,Y 453.532,Z 199.535,A -85,B 0,C 180,E1 -8395.713,E2 -8395.713} C_VEL
LIN {X 0,Y 453.904,Z 191.894,A -85,B 0,C 180,E1 -8399.19,E2 -8399.19} C_VEL
LIN {X 0,Y 454.261,Z 185.409,A -85,B 0,C 180,E1 -8402.258,E2 -8402.258} C_VEL
LIN {X 0,Y 454.541,Z 179.88,A -85,B 0,C 180,E1 -8404.968,E2 -8404.968} C_VEL
LIN {X 0,Y 454.27,Z 175.735,A -85,B 0,C 180,E1 -8407.109,E2 -8407.109} C_VEL
LIN {X 0,Y 453.51,Z 171,A -85,B 0,C 180,E1 -8409.733,E2 -8409.733} C_VEL
LIN {X 0,Y 453.48,Z 170.996,A -85,B 0,C 180,E1 -8412.99,E2 -8412.99} C_VEL
LIN {X 0,Y 453.452,Z 171.002,A -85,B 0,C 180,E1 -8415.777,E2 -8415.777} C_VEL
LIN {X 0,Y 453.464,Z 171,A -85,B 0,C 180,E1 -8418.207,E2 -8418.207} C_VEL
LIN {X 0,Y 453.455,Z 171.001,A -85,B 0,C 180,E1 -8420.795,E2 -8420.795} C_VEL
LIN {X 0,Y 453.439,Z 171.002,A -85,B 0,C 180,E1 -8423.916,E2 -8423.916} C_VEL
LIN {X 0,Y 453.464,Z 171.003,A -85,B 0,C 180,E1 -8427.15,E2 -8427.15} C_VEL
LIN {X 0,Y 453.454,Z 171,A -85,B 0,C 180,E1 -8430.267,E2 -8430.267} C_VEL
LIN {X 0,Y 453.484,Z 170.999,A -85,B 0,C 180,E1 -8433.293,E2 -8433.293} C_VEL
LIN {X 0,Y 453.493,Z 170.995,A -85,B 0,C 180,E1 -8436.238,E2 -8436.238} C_VEL
LIN {X 0,Y 453.494,Z 170.997,A -85,B 0,C 180,E1 -8439.118,E2 -8439.118} C_VEL
LIN {X 0,Y 453.495,Z 170.995,A -85,B 0,C 180,E1 -8441.944,E2 -8441.944} C_VEL
LIN {X 0,Y 453.523,Z 170.993,A -85,B 0,C 180,E1 -8444.726,E2 -8444.726} C_VEL
LIN {X 0,Y 453.576,Z 170.985,A -85,B 0,C 180,E1 -8447.472,E2 -8447.472} C_VEL
LIN {X 0,Y 453.577,Z 170.984,A -85,B 0,C 180,E1 -8451.086,E2 -8451.086} C_VEL
LIN {X 0,Y 453.675,Z 170.973,A -85,B 0,C 180,E1 -8453.775,E2 -8453.775} C_VEL
LIN {X 0,Y 453.717,Z 170.968,A -85,B 0,C 180,E1 -8457.337,E2 -8457.337} C_VEL
LIN {X 0,Y 453.791,Z 170.959,A -85,B 0,C 180,E1 -8460,E2 -8460} C_VEL
LIN {X 0,Y 453.748,Z 170.963,A -85,B 0,C 180,E1 -8462.664,E2 -8462.664} C_VEL
LIN {X 0,Y 453.658,Z 170.976,A -85,B 0,C 180,E1 -8466.226,E2 -8466.226} C_VEL
LIN {X 0,Y 453.566,Z 170.986,A -85,B 0,C 180,E1 -8468.914,E2 -8468.914} C_VEL
LIN {X 0,Y 453.538,Z 170.99,A -85,B 0,C 180,E1 -8472.53,E2 -8472.53} C_VEL
LIN {X 0,Y 453.533,Z 170.989,A -85,B 0,C 180,E1 -8476.197,E2 -8476.197} C_VEL
LIN {X 0,Y 453.5,Z 170.995,A -85,B 0,C 180,E1 -8479.043,E2 -8479.043} C_VEL
LIN {X 0,Y 453.455,Z 171.001,A -85,B 0,C 180,E1 -8481.838,E2 -8481.838} C_VEL
LIN {X 0,Y 453.492,Z 170.996,A -85,B 0,C 180,E1 -8484.736,E2 -8484.736} C_VEL
LIN {X 0,Y 453.513,Z 170.992,A -85,B 0,C 180,E1 -8487.961,E2 -8487.961} C_VEL
LIN {X 0,Y 453.465,Z 170.999,A -85,B 0,C 180,E1 -8490.761,E2 -8490.761} C_VEL
LIN {X 0,Y 453.46,Z 171,A -85,B 0,C 180,E1 -8493.915,E2 -8493.915} C_VEL
LIN {X 0,Y 453.437,Z 171.005,A -85,B 0,C 180,E1 -8497.192,E2 -8497.192} C_VEL
LIN {X 0,Y 453.471,Z 170.999,A -85,B 0,C 180,E1 -8499.452,E2 -8499.452} C_VEL
LIN {X 0,Y 453.464,Z 170.997,A -85,B 0,C 180,E1 -8501.937,E2 -8501.937} C_VEL
LIN {X 0,Y 453.475,Z 170.998,A -85,B 0,C 180,E1 -8505.473,E2 -8505.473} C_VEL
LIN {X 0,Y 453.47,Z 171.001,A -85,B 0,C 180,E1 -8508.211,E2 -8508.211} C_VEL
LIN {X 0,Y 453.43,Z 171.006,A -85,B 0,C 180,E1 -8510.804,E2 -8510.804} C_VEL
LIN {X 0,Y 453.348,Z 171.016,A -85,B 0,C 180,E1 -8512.245,E2 -8512.245} C_VEL
LIN {X 0,Y 453.361,Z 174.888,A -85,B 0,C 180,E1 -8515.247,E2 -8515.247} C_VEL
LIN {X 0,Y 453.211,Z 179.354,A -85,B 0,C 180,E1 -8518.529,E2 -8518.529} C_VEL
LIN {X 0,Y 453.081,Z 183.157,A -85,B 0,C 180,E1 -8521.26,E2 -8521.26} C_VEL
LIN {X 0,Y 452.953,Z 187.412,A -85,B 0,C 180,E1 -8524.251,E2 -8524.251} C_VEL
LIN {X 0,Y 452.832,Z 191.723,A -85,B 0,C 180,E1 -8527.171,E2 -8527.171} C_VEL
LIN {X 0,Y 452.739,Z 196.036,A -85,B 0,C 180,E1 -8530.032,E2 -8530.032} C_VEL
LIN {X 0,Y 452.706,Z 199.242,A -85,B 0,C 180,E1 -8532.117,E2 -8532.117} C_VEL
LIN {X 0,Y 455.576,Z 212.234,A -85,B 0,C 180,E1 -8532.612,E2 -8532.612} C_VEL
LIN {X 0,Y 456.572,Z 217.78,A -85,B 0,C 180,E1 -8532.872,E2 -8532.872} C_VEL
LIN {X 0,Y 456.178,Z 230.598,A -85,B 0,C 180,E1 -8533.515,E2 -8533.515} C_VEL
LIN {X 0,Y 455.615,Z 241.395,A -85,B 0,C 180,E1 -8534.225,E2 -8534.225} C_VEL
LIN {X 0,Y 454.994,Z 252.135,A -85,B 0,C 180,E1 -8535.12,E2 -8535.12} C_VEL
LIN {X 0,Y 454.524,Z 261.896,A -85,B 0,C 180,E1 -8536.134,E2 -8536.134} C_VEL
LIN {X 0,Y 454.015,Z 270.508,A -85,B 0,C 180,E1 -8537.221,E2 -8537.221} C_VEL
LIN {X 0,Y 453.894,Z 272.311,A -85,B 0,C 180,E1 -8537.473,E2 -8537.473} C_VEL
LIN {X 0,Y 453.005,Z 276.165,A -85,B 0,C 180,E1 -8538.028,E2 -8538.028} C_VEL
LIN {X 0,Y 449.855,Z 281.988,A -85,B 0,C 180,E1 -8538.966,E2 -8538.966} C_VEL
LIN {X 0,Y 446.75,Z 287.15,A -85,B 0,C 180,E1 -8539.975,E2 -8539.975} C_VEL
LIN {X 0,Y 445.944,Z 289.948,A -85,B 0,C 180,E1 -8540.636,E2 -8540.636} C_VEL
LIN {X 0,Y 445.685,Z 295.63,A -85,B 0,C 180,E1 -8542.297,E2 -8542.297} C_VEL
LIN {X 0,Y 445.534,Z 299.064,A -85,B 0,C 180,E1 -8543.66,E2 -8543.66} C_VEL
LIN {X 0,Y 445.476,Z 300.775,A -85,B 0,C 180,E1 -8544.568,E2 -8544.568} C_VEL
LIN {X 0,Y 445.409,Z 302.991,A -85,B 0,C 180,E1 -8546.381,E2 -8546.381} C_VEL
LIN {X 0,Y 445.437,Z 303.511,A -85,B 0,C 180,E1 -8547.287,E2 -8547.287} C_VEL
LIN {X 0,Y 445.343,Z 303.318,A -85,B 0,C 180,E1 -8549.095,E2 -8549.095} C_VEL
LIN {X 0,Y 445.378,Z 301.593,A -85,B 0,C 180,E1 -8550.903,E2 -8550.903} C_VEL
LIN {X 0,Y 445.455,Z 300.089,A -85,B 0,C 180,E1 -8551.807,E2 -8551.807} C_VEL
LIN {X 0,Y 445.633,Z 297.064,A -85,B 0,C 180,E1 -8553.163,E2 -8553.163} C_VEL
LIN {X 0,Y 445.783,Z 293,A -85,B 0,C 180,E1 -8554.52,E2 -8554.52} C_VEL
LIN {X 0,Y 446.045,Z 286.777,A -85,B 0,C 180,E1 -8556.104,E2 -8556.104} C_VEL
LIN {X 0,Y 446.446,Z 280.548,A -85,B 0,C 180,E1 -8557.359,E2 -8557.359} C_VEL
LIN {X 0,Y 446.795,Z 273.089,A -85,B 0,C 180,E1 -8558.593,E2 -8558.593} C_VEL
LIN {X 0,Y 447.355,Z 264.761,A -85,B 0,C 180,E1 -8559.722,E2 -8559.722} C_VEL
LIN {X 0,Y 447.944,Z 254.492,A -85,B 0,C 180,E1 -8560.851,E2 -8560.851} C_VEL
LIN {X 0,Y 448.475,Z 242.915,A -85,B 0,C 180,E1 -8561.868,E2 -8561.868} C_VEL
LIN {X 0,Y 448.974,Z 231.434,A -85,B 0,C 180,E1 -8562.657,E2 -8562.657} C_VEL
LIN {X 0,Y 449.52,Z 219.29,A -85,B 0,C 180,E1 -8563.283,E2 -8563.283} C_VEL
LIN {X 0,Y 447.244,Z 206.981,A -85,B 0,C 180,E1 -8563.832,E2 -8563.832} C_VEL
LIN {X 0,Y 445.61,Z 199.365,A -85,B 0,C 180,E1 -8564.119,E2 -8564.119} C_VEL
LIN {X 0,Y 445.728,Z 195.752,A -85,B 0,C 180,E1 -8566.486,E2 -8566.486} C_VEL
LIN {X 0,Y 445.767,Z 191.476,A -85,B 0,C 180,E1 -8569.333,E2 -8569.333} C_VEL
LIN {X 0,Y 445.884,Z 187.231,A -85,B 0,C 180,E1 -8572.225,E2 -8572.225} C_VEL
LIN {X 0,Y 445.966,Z 183.044,A -85,B 0,C 180,E1 -8575.179,E2 -8575.179} C_VEL
LIN {X 0,Y 446.125,Z 178.838,A -85,B 0,C 180,E1 -8578.2,E2 -8578.2} C_VEL
LIN {X 0,Y 446.271,Z 174.608,A -85,B 0,C 180,E1 -8581.308,E2 -8581.308} C_VEL
LIN {X 0,Y 446.277,Z 171.902,A -85,B 0,C 180,E1 -8583.445,E2 -8583.445} C_VEL
LIN {X 0,Y 446.389,Z 171.881,A -85,B 0,C 180,E1 -8585.625,E2 -8585.625} C_VEL
LIN {X 0,Y 446.412,Z 171.879,A -85,B 0,C 180,E1 -8589.026,E2 -8589.026} C_VEL
LIN {X 0,Y 446.421,Z 171.876,A -85,B 0,C 180,E1 -8592.275,E2 -8592.275} C_VEL
LIN {X 0,Y 446.44,Z 171.876,A -85,B 0,C 180,E1 -8595.1,E2 -8595.1} C_VEL
LIN {X 0,Y 446.425,Z 171.875,A -85,B 0,C 180,E1 -8598.608,E2 -8598.608} C_VEL
LIN {X 0,Y 446.45,Z 171.875,A -85,B 0,C 180,E1 -8600.973,E2 -8600.973} C_VEL
LIN {X 0,Y 446.395,Z 171.881,A -85,B 0,C 180,E1 -8604.371,E2 -8604.371} C_VEL
LIN {X 0,Y 446.397,Z 171.88,A -85,B 0,C 180,E1 -8607.636,E2 -8607.636} C_VEL
LIN {X 0,Y 446.443,Z 171.876,A -85,B 0,C 180,E1 -8610.79,E2 -8610.79} C_VEL
LIN {X 0,Y 446.449,Z 171.871,A -85,B 0,C 180,E1 -8613.846,E2 -8613.846} C_VEL
LIN {X 0,Y 446.419,Z 171.877,A -85,B 0,C 180,E1 -8616.822,E2 -8616.822} C_VEL
LIN {X 0,Y 446.428,Z 171.876,A -85,B 0,C 180,E1 -8619.736,E2 -8619.736} C_VEL
LIN {X 0,Y 446.432,Z 171.876,A -85,B 0,C 180,E1 -8622.596,E2 -8622.596} C_VEL
LIN {X 0,Y 446.486,Z 171.869,A -85,B 0,C 180,E1 -8625.413,E2 -8625.413} C_VEL
LIN {X 0,Y 446.533,Z 171.865,A -85,B 0,C 180,E1 -8628.193,E2 -8628.193} C_VEL
LIN {X 0,Y 446.573,Z 171.859,A -85,B 0,C 180,E1 -8631.857,E2 -8631.857} C_VEL
LIN {X 0,Y 446.627,Z 171.85,A -85,B 0,C 180,E1 -8634.582,E2 -8634.582} C_VEL
LIN {X 0,Y 446.674,Z 171.846,A -85,B 0,C 180,E1 -8637.294,E2 -8637.294} C_VEL
LIN {X 0,Y 446.753,Z 171.836,A -85,B 0,C 180,E1 -8640,E2 -8640} C_VEL
LIN {X 0,Y 446.684,Z 171.844,A -85,B 0,C 180,E1 -8642.705,E2 -8642.705} C_VEL
LIN {X 0,Y 446.626,Z 171.85,A -85,B 0,C 180,E1 -8646.324,E2 -8646.324} C_VEL
LIN {X 0,Y 446.558,Z 171.859,A -85,B 0,C 180,E1 -8649.055,E2 -8649.055} C_VEL
LIN {X 0,Y 446.501,Z 171.866,A -85,B 0,C 180,E1 -8652.73,E2 -8652.73} C_VEL
LIN {X 0,Y 446.456,Z 171.872,A -85,B 0,C 180,E1 -8656.46,E2 -8656.46} C_VEL
LIN {X 0,Y 446.437,Z 171.876,A -85,B 0,C 180,E1 -8659.305,E2 -8659.305} C_VEL
LIN {X 0,Y 446.412,Z 171.877,A -85,B 0,C 180,E1 -8662.2,E2 -8662.2} C_VEL
LIN {X 0,Y 446.446,Z 171.876,A -85,B 0,C 180,E1 -8665.153,E2 -8665.153} C_VEL
LIN {X 0,Y 446.456,Z 171.87,A -85,B 0,C 180,E1 -8668.181,E2 -8668.181} C_VEL
LIN {X 0,Y 446.391,Z 171.88,A -85,B 0,C 180,E1 -8671.302,E2 -8671.302} C_VEL
LIN {X 0,Y 446.403,Z 171.88,A -85,B 0,C 180,E1 -8674.525,E2 -8674.525} C_VEL
LIN {X 0,Y 446.414,Z 171.878,A -85,B 0,C 180,E1 -8678.085,E2 -8678.085} C_VEL
LIN {X 0,Y 446.426,Z 171.877,A -85,B 0,C 180,E1 -8680.923,E2 -8680.923} C_VEL
LIN {X 0,Y 446.425,Z 171.875,A -85,B 0,C 180,E1 -8683.843,E2 -8683.843} C_VEL
LIN {X 0,Y 446.428,Z 171.88,A -85,B 0,C 180,E1 -8686.4,E2 -8686.4} C_VEL
LIN {X 0,Y 446.441,Z 171.882,A -85,B 0,C 180,E1 -8689.806,E2 -8689.806} C_VEL
LIN {X 0,Y 446.516,Z 171.983,A -85,B 0,C 180,E1 -8690.64,E2 -8690.64} C_VEL
LIN {X 0,Y 447.38,Z 178.073,A -85,B 0,C 180,E1 -8693.911,E2 -8693.911} C_VEL
LIN {X 0,Y 447.284,Z 183.015,A -85,B 0,C 180,E1 -8696.384,E2 -8696.384} C_VEL
LIN {X 0,Y 446.951,Z 190.134,A -85,B 0,C 180,E1 -8699.793,E2 -8699.793} C_VEL
LIN {X 0,Y 446.521,Z 197.847,A -85,B 0,C 180,E1 -8703.351,E2 -8703.351} C_VEL
LIN {X 0,Y 446.258,Z 203.692,A -85,B 0,C 180,E1 -8705.984,E2 -8705.984} C_VEL
LIN {X 0,Y 446.075,Z 209.944,A -85,B 0,C 180,E1 -8708.756,E2 -8708.756} C_VEL
LIN {X 0,Y 445.808,Z 217.593,A -85,B 0,C 180,E1 -8712.099,E2 -8712.099} C_VEL
LIN {X 0,Y 445.705,Z 221.769,A -85,B 0,C 180,E1 -8713.919,E2 -8713.919} C_VEL
LIN {X 0,Y 447.878,Z 234.891,A -85,B 0,C 180,E1 -8714.357,E2 -8714.357} C_VEL
LIN {X 0,Y 449.159,Z 246.07,A -85,B 0,C 180,E1 -8714.866,E2 -8714.866} C_VEL
LIN {X 0,Y 448.607,Z 257.422,A -85,B 0,C 180,E1 -8715.485,E2 -8715.485} C_VEL
LIN {X 0,Y 448.024,Z 268.638,A -85,B 0,C 180,E1 -8716.277,E2 -8716.277} C_VEL
LIN {X 0,Y 447.592,Z 278.227,A -85,B 0,C 180,E1 -8717.121,E2 -8717.121} C_VEL
LIN {X 0,Y 447.006,Z 288.332,A -85,B 0,C 180,E1 -8718.208,E2 -8718.208} C_VEL
LIN {X 0,Y 446.468,Z 296.926,A -85,B 0,C 180,E1 -8719.343,E2 -8719.343} C_VEL
LIN {X 0,Y 446.073,Z 305.28,A -85,B 0,C 180,E1 -8720.708,E2 -8720.708} C_VEL
LIN {X 0,Y 445.735,Z 312.01,A -85,B 0,C 180,E1 -8722.071,E2 -8722.071} C_VEL
LIN {X 0,Y 445.528,Z 318.185,A -85,B 0,C 180,E1 -8723.661,E2 -8723.661} C_VEL
LIN {X 0,Y 445.475,Z 322.194,A -85,B 0,C 180,E1 -8725.023,E2 -8725.023} C_VEL
LIN {X 0,Y 445.378,Z 325.154,A -85,B 0,C 180,E1 -8726.382,E2 -8726.382} C_VEL
LIN {X 0,Y 445.432,Z 326.577,A -85,B 0,C 180,E1 -8727.288,E2 -8727.288} C_VEL
LIN {X 0,Y 445.338,Z 328.208,A -85,B 0,C 180,E1 -8729.096,E2 -8729.096} C_VEL
LIN {X 0,Y 445.343,Z 328.444,A -85,B 0,C 180,E1 -8730.001,E2 -8730.001} C_VEL
LIN {X 0,Y 445.338,Z 328.251,A -85,B 0,C 180,E1 -8730.905,E2 -8730.905} C_VEL
LIN {X 0,Y 445.432,Z 326.679,A -85,B 0,C 180,E1 -8732.713,E2 -8732.713} C_VEL
LIN {X 0,Y 445.378,Z 325.302,A -85,B 0,C 180,E1 -8733.619,E2 -8733.619} C_VEL
LIN {X 0,Y 445.474,Z 322.397,A -85,B 0,C 180,E1 -8734.978,E2 -8734.978} C_VEL
LIN {X 0,Y 445.574,Z 317.05,A -85,B 0,C 180,E1 -8736.748,E2 -8736.748} C_VEL
LIN {X 0,Y 445.793,Z 311.408,A -85,B 0,C 180,E1 -8738.157,E2 -8738.157} C_VEL
LIN {X 0,Y 446.155,Z 304.565,A -85,B 0,C 180,E1 -8739.52,E2 -8739.52} C_VEL
LIN {X 0,Y 446.585,Z 296.037,A -85,B 0,C 180,E1 -8740.885,E2 -8740.885} C_VEL
LIN {X 0,Y 447.18,Z 287.279,A -85,B 0,C 180,E1 -8742.019,E2 -8742.019} C_VEL
LIN {X 0,Y 447.714,Z 276.844,A -85,B 0,C 180,E1 -8743.123,E2 -8743.123} C_VEL
LIN {X 0,Y 448.368,Z 265.747,A -85,B 0,C 180,E1 -8744.061,E2 -8744.061} C_VEL
LIN {X 0,Y 449.06,Z 253.673,A -85,B 0,C 180,E1 -8744.849,E2 -8744.849} C_VEL
LIN {X 0,Y 449.315,Z 244.973,A -85,B 0,C 180,E1 -8745.304,E2 -8745.304} C_VEL
LIN {X 0,Y 447.56,Z 231.823,A -85,B 0,C 180,E1 -8745.886,E2 -8745.886} C_VEL
LIN {X 0,Y 445.722,Z 221.67,A -85,B 0,C 180,E1 -8746.243,E2 -8746.243} C_VEL
LIN {X 0,Y 445.904,Z 214.6,A -85,B 0,C 180,E1 -8749.328,E2 -8749.328} C_VEL
LIN {X 0,Y 446.174,Z 208.137,A -85,B 0,C 180,E1 -8752.211,E2 -8752.211} C_VEL
LIN {X 0,Y 446.467,Z 200.51,A -85,B 0,C 180,E1 -8755.65,E2 -8755.65} C_VEL
LIN {X 0,Y 446.873,Z 192.899,A -85,B 0,C 180,E1 -8759.177,E2 -8759.177} C_VEL
LIN {X 0,Y 447.252,Z 186.412,A -85,B 0,C 180,E1 -8762.292,E2 -8762.292} C_VEL
LIN {X 0,Y 447.578,Z 179.968,A -85,B 0,C 180,E1 -8765.518,E2 -8765.518} C_VEL
LIN {X 0,Y 446.988,Z 175.049,A -85,B 0,C 180,E1 -8768.173,E2 -8768.173} C_VEL
LIN {X 0,Y 446.47,Z 171.877,A -85,B 0,C 180,E1 -8770.01,E2 -8770.01} C_VEL
LIN {X 0,Y 446.435,Z 171.878,A -85,B 0,C 180,E1 -8773.601,E2 -8773.601} C_VEL
LIN {X 0,Y 446.386,Z 171.883,A -85,B 0,C 180,E1 -8776.402,E2 -8776.402} C_VEL
LIN {X 0,Y 446.412,Z 171.879,A -85,B 0,C 180,E1 -8779.081,E2 -8779.081} C_VEL
LIN {X 0,Y 446.391,Z 171.88,A -85,B 0,C 180,E1 -8782.119,E2 -8782.119} C_VEL
LIN {X 0,Y 446.412,Z 171.88,A -85,B 0,C 180,E1 -8785.475,E2 -8785.475} C_VEL
LIN {X 0,Y 446.396,Z 171.88,A -85,B 0,C 180,E1 -8788.698,E2 -8788.698} C_VEL
LIN {X 0,Y 446.464,Z 171.872,A -85,B 0,C 180,E1 -8791.82,E2 -8791.82} C_VEL
LIN {X 0,Y 446.438,Z 171.875,A -85,B 0,C 180,E1 -8794.847,E2 -8794.847} C_VEL
LIN {X 0,Y 446.462,Z 171.869,A -85,B 0,C 180,E1 -8798.232,E2 -8798.232} C_VEL
LIN {X 0,Y 446.439,Z 171.874,A -85,B 0,C 180,E1 -8801.649,E2 -8801.649} C_VEL
LIN {X 0,Y 446.49,Z 171.87,A -85,B 0,C 180,E1 -8804.479,E2 -8804.479} C_VEL
LIN {X 0,Y 446.518,Z 171.865,A -85,B 0,C 180,E1 -8808.193,E2 -8808.193} C_VEL
LIN {X 0,Y 446.577,Z 171.856,A -85,B 0,C 180,E1 -8811.858,E2 -8811.858} C_VEL
LIN {X 0,Y 446.635,Z 171.851,A -85,B 0,C 180,E1 -8814.583,E2 -8814.583} C_VEL
LIN {X 0,Y 446.634,Z 171.851,A -85,B 0,C 180,E1 -8818.197,E2 -8818.197} C_VEL
LIN {X 0,Y 446.761,Z 171.835,A -85,B 0,C 180,E1 -8820,E2 -8820} C_VEL
LIN {X 0,Y 446.693,Z 171.842,A -85,B 0,C 180,E1 -8822.706,E2 -8822.706} C_VEL
LIN {X 0,Y 446.626,Z 171.851,A -85,B 0,C 180,E1 -8826.324,E2 -8826.324} C_VEL
LIN {X 0,Y 446.512,Z 171.865,A -85,B 0,C 180,E1 -8829.056,E2 -8829.056} C_VEL
LIN {X 0,Y 446.496,Z 171.866,A -85,B 0,C 180,E1 -8832.731,E2 -8832.731} C_VEL
LIN {X 0,Y 446.476,Z 171.867,A -85,B 0,C 180,E1 -8836.46,E2 -8836.46} C_VEL
LIN {X 0,Y 446.448,Z 171.876,A -85,B 0,C 180,E1 -8839.304,E2 -8839.304} C_VEL
LIN {X 0,Y 446.397,Z 171.88,A -85,B 0,C 180,E1 -8842.201,E2 -8842.201} C_VEL
LIN {X 0,Y 446.436,Z 171.876,A -85,B 0,C 180,E1 -8845.154,E2 -8845.154} C_VEL
LIN {X 0,Y 446.466,Z 171.869,A -85,B 0,C 180,E1 -8848.18,E2 -8848.18} C_VEL
LIN {X 0,Y 446.401,Z 171.881,A -85,B 0,C 180,E1 -8851.302,E2 -8851.302} C_VEL
LIN {X 0,Y 446.413,Z 171.878,A -85,B 0,C 180,E1 -8854.525,E2 -8854.525} C_VEL
LIN {X 0,Y 446.399,Z 171.879,A -85,B 0,C 180,E1 -8858.081,E2 -8858.081} C_VEL
LIN {X 0,Y 446.414,Z 171.881,A -85,B 0,C 180,E1 -8860.92,E2 -8860.92} C_VEL
LIN {X 0,Y 446.39,Z 171.878,A -85,B 0,C 180,E1 -8863.848,E2 -8863.848} C_VEL
LIN {X 0,Y 446.388,Z 171.884,A -85,B 0,C 180,E1 -8866.406,E2 -8866.406} C_VEL
LIN {X 0,Y 446.419,Z 171.878,A -85,B 0,C 180,E1 -8869.084,E2 -8869.084} C_VEL
LIN {X 0,Y 446.324,Z 171.891,A -85,B 0,C 180,E1 -8872.115,E2 -8872.115} C_VEL
LIN {X 0,Y 446.321,Z 175.422,A -85,B 0,C 180,E1 -8874.968,E2 -8874.968} C_VEL
LIN {X 0,Y 446.185,Z 178.97,A -85,B 0,C 180,E1 -8877.621,E2 -8877.621} C_VEL
LIN {X 0,Y 446.037,Z 183.26,A -85,B 0,C 180,E1 -8880.763,E2 -8880.763} C_VEL
LIN {X 0,Y 445.892,Z 187.727,A -85,B 0,C 180,E1 -8883.952,E2 -8883.952} C_VEL
LIN {X 0,Y 445.793,Z 191.853,A -85,B 0,C 180,E1 -8886.789,E2 -8886.789} C_VEL
LIN {X 0,Y 445.67,Z 196.199,A -85,B 0,C 180,E1 -8889.701,E2 -8889.701} C_VEL
LIN {X 0,Y 445.652,Z 199.391,A -85,B 0,C 180,E1 -8891.824,E2 -8891.824} C_VEL
LIN {X 0,Y 449.005,Z 214.899,A -85,B 0,C 180,E1 -8892.465,E2 -8892.465} C_VEL
LIN {X 0,Y 449.732,Z 220.301,A -85,B 0,C 180,E1 -8892.728,E2 -8892.728} C_VEL
LIN {X 0,Y 449.264,Z 232.347,A -85,B 0,C 180,E1 -8893.37,E2 -8893.37} C_VEL
LIN {X 0,Y 448.613,Z 244.216,A -85,B 0,C 180,E1 -8894.205,E2 -8894.205} C_VEL
LIN {X 0,Y 448.022,Z 254.468,A -85,B 0,C 180,E1 -8895.116,E2 -8895.116} C_VEL
LIN {X 0,Y 447.499,Z 263.867,A -85,B 0,C 180,E1 -8896.143,E2 -8896.143} C_VEL
LIN {X 0,Y 446.886,Z 272.932,A -85,B 0,C 180,E1 -8897.359,E2 -8897.359} C_VEL
LIN {X 0,Y 446.557,Z 280.724,A -85,B 0,C 180,E1 -8898.655,E2 -8898.655} C_VEL
LIN {X 0,Y 446.085,Z 287.402,A -85,B 0,C 180,E1 -8900.02,E2 -8900.02} C_VEL
LIN {X 0,Y 445.944,Z 289.948,A -85,B 0,C 180,E1 -8900.636,E2 -8900.636} C_VEL
LIN {X 0,Y 445.145,Z 292.54,A -85,B 0,C 180,E1 -8901.313,E2 -8901.313} C_VEL
LIN {X 0,Y 442.1,Z 296.247,A -85,B 0,C 180,E1 -8902.436,E2 -8902.436} C_VEL
LIN {X 0,Y 439.581,Z 298.717,A -85,B 0,C 180,E1 -8903.366,E2 -8903.366} C_VEL
LIN {X 0,Y 438.495,Z 300.266,A -85,B 0,C 180,E1 -8904.099,E2 -8904.099} C_VEL
LIN {X 0,Y 438.402,Z 300.696,A -85,B 0,C 180,E1 -8904.349,E2 -8904.349} C_VEL
LIN {X 0,Y 438.322,Z 302.251,A -85,B 0,C 180,E1 -8905.401,E2 -8905.401} C_VEL
LIN {X 0,Y 438.364,Z 303.701,A -85,B 0,C 180,E1 -8907.243,E2 -8907.243} C_VEL
LIN {X 0,Y 438.256,Z 303.526,A -85,B 0,C 180,E1 -8909.081,E2 -8909.081} C_VEL
LIN {X 0,Y 438.29,Z 301.818,A -85,B 0,C 180,E1 -8910.918,E2 -8910.918} C_VEL
LIN {X 0,Y 438.374,Z 300.327,A -85,B 0,C 180,E1 -8911.837,E2 -8911.837} C_VEL
LIN {X 0,Y 438.563,Z 297.317,A -85,B 0,C 180,E1 -8913.214,E2 -8913.214} C_VEL
LIN {X 0,Y 438.709,Z 293.27,A -85,B 0,C 180,E1 -8914.593,E2 -8914.593} C_VEL
LIN {X 0,Y 439.013,Z 287.064,A -85,B 0,C 180,E1 -8916.202,E2 -8916.202} C_VEL
LIN {X 0,Y 439.397,Z 281.282,A -85,B 0,C 180,E1 -8917.397,E2 -8917.397} C_VEL
LIN {X 0,Y 439.802,Z 273.418,A -85,B 0,C 180,E1 -8918.731,E2 -8918.731} C_VEL
LIN {X 0,Y 440.364,Z 265.118,A -85,B 0,C 180,E1 -8919.877,E2 -8919.877} C_VEL
LIN {X 0,Y 441,Z 254.898,A -85,B 0,C 180,E1 -8921.024,E2 -8921.024} C_VEL
LIN {X 0,Y 441.56,Z 243.365,A -85,B 0,C 180,E1 -8922.056,E2 -8922.056} C_VEL
LIN {X 0,Y 442.089,Z 231.968,A -85,B 0,C 180,E1 -8922.858,E2 -8922.858} C_VEL
LIN {X 0,Y 442.63,Z 219.948,A -85,B 0,C 180,E1 -8923.494,E2 -8923.494} C_VEL
LIN {X 0,Y 440.133,Z 206.865,A -85,B 0,C 180,E1 -8924.092,E2 -8924.092} C_VEL
LIN {X 0,Y 438.552,Z 199.574,A -85,B 0,C 180,E1 -8924.354,E2 -8924.354} C_VEL
LIN {X 0,Y 438.644,Z 195.977,A -85,B 0,C 180,E1 -8926.76,E2 -8926.76} C_VEL
LIN {X 0,Y 438.701,Z 191.675,A -85,B 0,C 180,E1 -8929.657,E2 -8929.657} C_VEL
LIN {X 0,Y 438.834,Z 187.419,A -85,B 0,C 180,E1 -8932.602,E2 -8932.602} C_VEL
LIN {X 0,Y 438.926,Z 183.228,A -85,B 0,C 180,E1 -8935.612,E2 -8935.612} C_VEL
LIN {X 0,Y 439.082,Z 179.002,A -85,B 0,C 180,E1 -8938.694,E2 -8938.694} C_VEL
LIN {X 0,Y 439.233,Z 174.574,A -85,B 0,C 180,E1 -8942.001,E2 -8942.001} C_VEL
LIN {X 0,Y 439.223,Z 173.337,A -85,B 0,C 180,E1 -8942.955,E2 -8942.955} C_VEL
LIN {X 0,Y 439.254,Z 172.773,A -85,B 0,C 180,E1 -8944.052,E2 -8944.052} C_VEL
LIN {X 0,Y 439.334,Z 172.76,A -85,B 0,C 180,E1 -8946.884,E2 -8946.884} C_VEL
LIN {X 0,Y 439.389,Z 172.755,A -85,B 0,C 180,E1 -8949.846,E2 -8949.846} C_VEL
LIN {X 0,Y 439.37,Z 172.755,A -85,B 0,C 180,E1 -8952.625,E2 -8952.625} C_VEL
LIN {X 0,Y 439.385,Z 172.751,A -85,B 0,C 180,E1 -8956.031,E2 -8956.031} C_VEL
LIN {X 0,Y 439.382,Z 172.757,A -85,B 0,C 180,E1 -8959.019,E2 -8959.019} C_VEL
LIN {X 0,Y 439.361,Z 172.756,A -85,B 0,C 180,E1 -8961.604,E2 -8961.604} C_VEL
LIN {X 0,Y 439.375,Z 172.756,A -85,B 0,C 180,E1 -8964.841,E2 -8964.841} C_VEL
LIN {X 0,Y 439.348,Z 172.758,A -85,B 0,C 180,E1 -8968.137,E2 -8968.137} C_VEL
LIN {X 0,Y 439.398,Z 172.751,A -85,B 0,C 180,E1 -8971.325,E2 -8971.325} C_VEL
LIN {X 0,Y 439.387,Z 172.754,A -85,B 0,C 180,E1 -8974.414,E2 -8974.414} C_VEL
LIN {X 0,Y 439.355,Z 172.755,A -85,B 0,C 180,E1 -8977.424,E2 -8977.424} C_VEL
LIN {X 0,Y 439.41,Z 172.75,A -85,B 0,C 180,E1 -8980.661,E2 -8980.661} C_VEL
LIN {X 0,Y 439.443,Z 172.747,A -85,B 0,C 180,E1 -8984.223,E2 -8984.223} C_VEL
LIN {X 0,Y 439.494,Z 172.74,A -85,B 0,C 180,E1 -8988.001,E2 -8988.001} C_VEL
LIN {X 0,Y 439.51,Z 172.736,A -85,B 0,C 180,E1 -8990.798,E2 -8990.798} C_VEL
LIN {X 0,Y 439.604,Z 172.726,A -85,B 0,C 180,E1 -8993.574,E2 -8993.574} C_VEL
LIN {X 0,Y 439.621,Z 172.724,A -85,B 0,C 180,E1 -8997.251,E2 -8997.251} C_VEL
LIN {X 0,Y 439.724,Z 172.712,A -85,B 0,C 180,E1 -9000,E2 -9000} C_VEL
LIN {X 0,Y 439.631,Z 172.722,A -85,B 0,C 180,E1 -9002.749,E2 -9002.749} C_VEL
LIN {X 0,Y 439.595,Z 172.726,A -85,B 0,C 180,E1 -9006.425,E2 -9006.425} C_VEL
LIN {X 0,Y 439.506,Z 172.739,A -85,B 0,C 180,E1 -9009.201,E2 -9009.201} C_VEL
LIN {X 0,Y 439.471,Z 172.742,A -85,B 0,C 180,E1 -9012.728,E2 -9012.728} C_VEL
LIN {X 0,Y 439.413,Z 172.749,A -85,B 0,C 180,E1 -9016.349,E2 -9016.349} C_VEL
LIN {X 0,Y 439.402,Z 172.752,A -85,B 0,C 180,E1 -9019.626,E2 -9019.626} C_VEL
LIN {X 0,Y 439.354,Z 172.757,A -85,B 0,C 180,E1 -9022.576,E2 -9022.576} C_VEL
LIN {X 0,Y 439.385,Z 172.752,A -85,B 0,C 180,E1 -9025.586,E2 -9025.586} C_VEL
LIN {X 0,Y 439.397,Z 172.754,A -85,B 0,C 180,E1 -9028.675,E2 -9028.675} C_VEL
LIN {X 0,Y 439.346,Z 172.757,A -85,B 0,C 180,E1 -9031.863,E2 -9031.863} C_VEL
LIN {X 0,Y 439.374,Z 172.756,A -85,B 0,C 180,E1 -9035.158,E2 -9035.158} C_VEL
LIN {X 0,Y 439.375,Z 172.756,A -85,B 0,C 180,E1 -9038.596,E2 -9038.596} C_VEL
LIN {X 0,Y 439.384,Z 172.752,A -85,B 0,C 180,E1 -9041.262,E2 -9041.262} C_VEL
LIN {X 0,Y 439.391,Z 172.752,A -85,B 0,C 180,E1 -9044.731,E2 -9044.731} C_VEL
LIN {X 0,Y 439.387,Z 172.757,A -85,B 0,C 180,E1 -9047.799,E2 -9047.799} C_VEL
LIN {X 0,Y 439.444,Z 172.777,A -85,B 0,C 180,E1 -9050.382,E2 -9050.382} C_VEL
LIN {X 0,Y 440.373,Z 179.058,A -85,B 0,C 180,E1 -9053.812,E2 -9053.812} C_VEL
LIN {X 0,Y 440.286,Z 183.524,A -85,B 0,C 180,E1 -9056.103,E2 -9056.103} C_VEL
LIN {X 0,Y 439.919,Z 190.727,A -85,B 0,C 180,E1 -9059.62,E2 -9059.62} C_VEL
LIN {X 0,Y 439.463,Z 198.78,A -85,B 0,C 180,E1 -9063.401,E2 -9063.401} C_VEL
LIN {X 0,Y 439.162,Z 205.376,A -85,B 0,C 180,E1 -9066.419,E2 -9066.419} C_VEL
LIN {X 0,Y 438.923,Z 211.941,A -85,B 0,C 180,E1 -9069.376,E2 -9069.376} C_VEL
LIN {X 0,Y 438.672,Z 219.538,A -85,B 0,C 180,E1 -9072.761,E2 -9072.761} C_VEL
LIN {X 0,Y 438.621,Z 221.575,A -85,B 0,C 180,E1 -9073.664,E2 -9073.664} C_VEL
LIN {X 0,Y 440.784,Z 234.812,A -85,B 0,C 180,E1 -9074.115,E2 -9074.115} C_VEL
LIN {X 0,Y 442.256,Z 245.648,A -85,B 0,C 180,E1 -9074.624,E2 -9074.624} C_VEL
LIN {X 0,Y 441.714,Z 257.052,A -85,B 0,C 180,E1 -9075.254,E2 -9075.254} C_VEL
LIN {X 0,Y 441.118,Z 268.302,A -85,B 0,C 180,E1 -9076.058,E2 -9076.058} C_VEL
LIN {X 0,Y 440.597,Z 278.332,A -85,B 0,C 180,E1 -9076.954,E2 -9076.954} C_VEL
LIN {X 0,Y 440.039,Z 288.04,A -85,B 0,C 180,E1 -9078.018,E2 -9078.018} C_VEL
LIN {X 0,Y 439.466,Z 296.655,A -85,B 0,C 180,E1 -9079.171,E2 -9079.171} C_VEL
LIN {X 0,Y 439.041,Z 305.023,A -85,B 0,C 180,E1 -9080.558,E2 -9080.558} C_VEL
LIN {X 0,Y 438.683,Z 311.765,A -85,B 0,C 180,E1 -9081.943,E2 -9081.943} C_VEL
LIN {X 0,Y 438.442,Z 318.184,A -85,B 0,C 180,E1 -9083.632,E2 -9083.632} C_VEL
LIN {X 0,Y 438.384,Z 321.97,A -85,B 0,C 180,E1 -9084.942,E2 -9084.942} C_VEL
LIN {X 0,Y 438.28,Z 324.936,A -85,B 0,C 180,E1 -9086.323,E2 -9086.323} C_VEL
LIN {X 0,Y 438.34,Z 326.366,A -85,B 0,C 180,E1 -9087.244,E2 -9087.244} C_VEL
LIN {X 0,Y 438.252,Z 328.005,A -85,B 0,C 180,E1 -9089.082,E2 -9089.082} C_VEL
LIN {X 0,Y 438.254,Z 328.245,A -85,B 0,C 180,E1 -9090.001,E2 -9090.001} C_VEL
LIN {X 0,Y 438.252,Z 328.059,A -85,B 0,C 180,E1 -9090.919,E2 -9090.919} C_VEL
LIN {X 0,Y 438.34,Z 326.494,A -85,B 0,C 180,E1 -9092.757,E2 -9092.757} C_VEL
LIN {X 0,Y 438.279,Z 325.121,A -85,B 0,C 180,E1 -9093.678,E2 -9093.678} C_VEL
LIN {X 0,Y 438.383,Z 322.223,A -85,B 0,C 180,E1 -9095.059,E2 -9095.059} C_VEL
LIN {X 0,Y 438.448,Z 318.295,A -85,B 0,C 180,E1 -9096.443,E2 -9096.443} C_VEL
LIN {X 0,Y 438.662,Z 313.241,A -85,B 0,C 180,E1 -9097.827,E2 -9097.827} C_VEL
LIN {X 0,Y 438.986,Z 306.892,A -85,B 0,C 180,E1 -9099.212,E2 -9099.212} C_VEL
LIN {X 0,Y 439.399,Z 298.949,A -85,B 0,C 180,E1 -9100.599,E2 -9100.599} C_VEL
LIN {X 0,Y 440.034,Z 290.87,A -85,B 0,C 180,E1 -9101.749,E2 -9101.749} C_VEL
LIN {X 0,Y 440.591,Z 281.019,A -85,B 0,C 180,E1 -9102.904,E2 -9102.904} C_VEL
LIN {X 0,Y 441.13,Z 271.355,A -85,B 0,C 180,E1 -9103.826,E2 -9103.826} C_VEL
LIN {X 0,Y 441.765,Z 260.949,A -85,B 0,C 180,E1 -9104.628,E2 -9104.628} C_VEL
LIN {X 0,Y 442.443,Z 248.446,A -85,B 0,C 180,E1 -9105.371,E2 -9105.371} C_VEL
LIN {X 0,Y 442.074,Z 242.435,A -85,B 0,C 180,E1 -9105.679,E2 -9105.679} C_VEL
LIN {X 0,Y 440.218,Z 229.733,A -85,B 0,C 180,E1 -9106.232,E2 -9106.232} C_VEL
LIN {X 0,Y 438.649,Z 221.488,A -85,B 0,C 180,E1 -9106.513,E2 -9106.513} C_VEL
LIN {X 0,Y 438.847,Z 214.459,A -85,B 0,C 180,E1 -9109.651,E2 -9109.651} C_VEL
LIN {X 0,Y 439.155,Z 208.008,A -85,B 0,C 180,E1 -9112.586,E2 -9112.586} C_VEL
LIN {X 0,Y 439.403,Z 201.494,A -85,B 0,C 180,E1 -9115.584,E2 -9115.584} C_VEL
LIN {X 0,Y 439.852,Z 193.887,A -85,B 0,C 180,E1 -9119.164,E2 -9119.164} C_VEL
LIN {X 0,Y 440.201,Z 187.67,A -85,B 0,C 180,E1 -9122.203,E2 -9122.203} C_VEL
LIN {X 0,Y 440.518,Z 182.046,A -85,B 0,C 180,E1 -9125.051,E2 -9125.051} C_VEL
LIN {X 0,Y 440.227,Z 177.792,A -85,B 0,C 180,E1 -9127.345,E2 -9127.345} C_VEL
LIN {X 0,Y 439.421,Z 172.755,A -85,B 0,C 180,E1 -9130.228,E2 -9130.228} C_VEL
LIN {X 0,Y 439.382,Z 172.755,A -85,B 0,C 180,E1 -9133.453,E2 -9133.453} C_VEL
LIN {X 0,Y 439.338,Z 172.762,A -85,B 0,C 180,E1 -9136.539,E2 -9136.539} C_VEL
LIN {X 0,Y 439.365,Z 172.756,A -85,B 0,C 180,E1 -9139.018,E2 -9139.018} C_VEL
LIN {X 0,Y 439.353,Z 172.76,A -85,B 0,C 180,E1 -9141.607,E2 -9141.607} C_VEL
LIN {X 0,Y 439.383,Z 172.752,A -85,B 0,C 180,E1 -9144.843,E2 -9144.843} C_VEL
LIN {X 0,Y 439.353,Z 172.756,A -85,B 0,C 180,E1 -9148.138,E2 -9148.138} C_VEL
LIN {X 0,Y 439.412,Z 172.751,A -85,B 0,C 180,E1 -9151.597,E2 -9151.597} C_VEL
LIN {X 0,Y 439.385,Z 172.753,A -85,B 0,C 180,E1 -9154.414,E2 -9154.414} C_VEL
LIN {X 0,Y 439.362,Z 172.755,A -85,B 0,C 180,E1 -9157.424,E2 -9157.424} C_VEL
LIN {X 0,Y 439.419,Z 172.752,A -85,B 0,C 180,E1 -9160.661,E2 -9160.661} C_VEL
LIN {X 0,Y 439.45,Z 172.746,A -85,B 0,C 180,E1 -9164.224,E2 -9164.224} C_VEL
LIN {X 0,Y 439.485,Z 172.741,A -85,B 0,C 180,E1 -9168.001,E2 -9168.001} C_VEL
LIN {X 0,Y 439.525,Z 172.733,A -85,B 0,C 180,E1 -9171.726,E2 -9171.726} C_VEL
LIN {X 0,Y 439.611,Z 172.726,A -85,B 0,C 180,E1 -9174.496,E2 -9174.496} C_VEL
LIN {X 0,Y 439.605,Z 172.727,A -85,B 0,C 180,E1 -9178.168,E2 -9178.168} C_VEL
LIN {X 0,Y 439.731,Z 172.711,A -85,B 0,C 180,E1 -9180,E2 -9180} C_VEL
LIN {X 0,Y 439.64,Z 172.72,A -85,B 0,C 180,E1 -9182.749,E2 -9182.749} C_VEL
LIN {X 0,Y 439.596,Z 172.727,A -85,B 0,C 180,E1 -9186.426,E2 -9186.426} C_VEL
LIN {X 0,Y 439.474,Z 172.742,A -85,B 0,C 180,E1 -9189.202,E2 -9189.202} C_VEL
LIN {X 0,Y 439.441,Z 172.745,A -85,B 0,C 180,E1 -9192.939,E2 -9192.939} C_VEL
LIN {X 0,Y 439.439,Z 172.744,A -85,B 0,C 180,E1 -9196.357,E2 -9196.357} C_VEL
LIN {X 0,Y 439.381,Z 172.755,A -85,B 0,C 180,E1 -9199.628,E2 -9199.628} C_VEL
LIN {X 0,Y 439.344,Z 172.757,A -85,B 0,C 180,E1 -9202.577,E2 -9202.577} C_VEL
LIN {X 0,Y 439.385,Z 172.756,A -85,B 0,C 180,E1 -9205.587,E2 -9205.587} C_VEL
LIN {X 0,Y 439.406,Z 172.749,A -85,B 0,C 180,E1 -9208.675,E2 -9208.675} C_VEL
LIN {X 0,Y 439.356,Z 172.756,A -85,B 0,C 180,E1 -9211.862,E2 -9211.862} C_VEL
LIN {X 0,Y 439.384,Z 172.755,A -85,B 0,C 180,E1 -9215.158,E2 -9215.158} C_VEL
LIN {X 0,Y 439.363,Z 172.757,A -85,B 0,C 180,E1 -9218.598,E2 -9218.598} C_VEL
LIN {X 0,Y 439.376,Z 172.754,A -85,B 0,C 180,E1 -9221.259,E2 -9221.259} C_VEL
LIN {X 0,Y 439.39,Z 172.755,A -85,B 0,C 180,E1 -9224.731,E2 -9224.731} C_VEL
LIN {X 0,Y 439.387,Z 172.752,A -85,B 0,C 180,E1 -9227.798,E2 -9227.798} C_VEL
LIN {X 0,Y 439.351,Z 172.759,A -85,B 0,C 180,E1 -9230.222,E2 -9230.222} C_VEL
LIN {X 0,Y 439.32,Z 172.765,A -85,B 0,C 180,E1 -9231.617,E2 -9231.617} C_VEL
LIN {X 0,Y 439.276,Z 173.262,A -85,B 0,C 180,E1 -9232.56,E2 -9232.56} C_VEL
LIN {X 0,Y 439.298,Z 176.159,A -85,B 0,C 180,E1 -9234.837,E2 -9234.837} C_VEL
LIN {X 0,Y 439.134,Z 180.49,A -85,B 0,C 180,E1 -9238.122,E2 -9238.122} C_VEL
LIN {X 0,Y 438.967,Z 184.793,A -85,B 0,C 180,E1 -9241.296,E2 -9241.296} C_VEL
LIN {X 0,Y 438.801,Z 189.076,A -85,B 0,C 180,E1 -9244.379,E2 -9244.379} C_VEL
LIN {X 0,Y 438.752,Z 191.984,A -85,B 0,C 180,E1 -9246.395,E2 -9246.395} C_VEL
LIN {X 0,Y 438.601,Z 196.341,A -85,B 0,C 180,E1 -9249.359,E2 -9249.359} C_VEL
LIN {X 0,Y 438.57,Z 199.698,A -85,B 0,C 180,E1 -9251.565,E2 -9251.565} C_VEL
LIN {X 0,Y 441.637,Z 213.148,A -85,B 0,C 180,E1 -9252.108,E2 -9252.108} C_VEL
LIN {X 0,Y 442.875,Z 221.422,A -85,B 0,C 180,E1 -9252.516,E2 -9252.516} C_VEL
LIN {X 0,Y 442.366,Z 233.816,A -85,B 0,C 180,E1 -9253.21,E2 -9253.21} C_VEL
LIN {X 0,Y 441.67,Z 245.588,A -85,B 0,C 180,E1 -9254.069,E2 -9254.069} C_VEL
LIN {X 0,Y 441.038,Z 256.739,A -85,B 0,C 180,E1 -9255.111,E2 -9255.111} C_VEL
LIN {X 0,Y 440.445,Z 265.737,A -85,B 0,C 180,E1 -9256.152,E2 -9256.152} C_VEL
LIN {X 0,Y 439.808,Z 274.528,A -85,B 0,C 180,E1 -9257.394,E2 -9257.394} C_VEL
LIN {X 0,Y 439.467,Z 282.041,A -85,B 0,C 180,E1 -9258.703,E2 -9258.703} C_VEL
LIN {X 0,Y 439.037,Z 287.51,A -85,B 0,C 180,E1 -9259.858,E2 -9259.858} C_VEL
LIN {X 0,Y 438.76,Z 292.848,A -85,B 0,C 180,E1 -9261.247,E2 -9261.247} C_VEL
LIN {X 0,Y 438.541,Z 297.011,A -85,B 0,C 180,E1 -9262.634,E2 -9262.634} C_VEL
LIN {X 0,Y 438.467,Z 299.321,A -85,B 0,C 180,E1 -9263.607,E2 -9263.607} C_VEL
LIN {X 0,Y 438.402,Z 300.696,A -85,B 0,C 180,E1 -9264.349,E2 -9264.349} C_VEL
LIN {X 0,Y 437.715,Z 301.954,A -85,B 0,C 180,E1 -9265.098,E2 -9265.098} C_VEL
LIN {X 0,Y 434.828,Z 303.398,A -85,B 0,C 180,E1 -9266.329,E2 -9266.329} C_VEL
LIN {X 0,Y 432.377,Z 303.948,A -85,B 0,C 180,E1 -9267.332,E2 -9267.332} C_VEL
LIN {X 0,Y 431.299,Z 304.009,A -85,B 0,C 180,E1 -9268.108,E2 -9268.108} C_VEL
LIN {X 0,Y 431.198,Z 303.937,A -85,B 0,C 180,E1 -9268.371,E2 -9268.371} C_VEL
LIN {X 0,Y 431.172,Z 303.08,A -85,B 0,C 180,E1 -9269.999,E2 -9269.999} C_VEL
LIN {X 0,Y 431.206,Z 302.043,A -85,B 0,C 180,E1 -9270.933,E2 -9270.933} C_VEL
LIN {X 0,Y 431.295,Z 300.564,A -85,B 0,C 180,E1 -9271.867,E2 -9271.867} C_VEL
LIN {X 0,Y 431.496,Z 297.569,A -85,B 0,C 180,E1 -9273.267,E2 -9273.267} C_VEL
LIN {X 0,Y 431.635,Z 293.539,A -85,B 0,C 180,E1 -9274.669,E2 -9274.669} C_VEL
LIN {X 0,Y 431.984,Z 287.35,A -85,B 0,C 180,E1 -9276.304,E2 -9276.304} C_VEL
LIN {X 0,Y 432.406,Z 280.614,A -85,B 0,C 180,E1 -9277.705,E2 -9277.705} C_VEL
LIN {X 0,Y 432.803,Z 273.746,A -85,B 0,C 180,E1 -9278.873,E2 -9278.873} C_VEL
LIN {X 0,Y 433.391,Z 265.472,A -85,B 0,C 180,E1 -9280.038,E2 -9280.038} C_VEL
LIN {X 0,Y 434.047,Z 255.301,A -85,B 0,C 180,E1 -9281.202,E2 -9281.202} C_VEL
LIN {X 0,Y 434.655,Z 243.81,A -85,B 0,C 180,E1 -9282.251,E2 -9282.251} C_VEL
LIN {X 0,Y 435.201,Z 232.484,A -85,B 0,C 180,E1 -9283.065,E2 -9283.065} C_VEL
LIN {X 0,Y 435.708,Z 220.602,A -85,B 0,C 180,E1 -9283.712,E2 -9283.712} C_VEL
LIN {X 0,Y 433.202,Z 207.704,A -85,B 0,C 180,E1 -9284.322,E2 -9284.322} C_VEL
LIN {X 0,Y 431.506,Z 199.769,A -85,B 0,C 180,E1 -9284.621,E2 -9284.621} C_VEL
LIN {X 0,Y 431.583,Z 196.172,A -85,B 0,C 180,E1 -9287.043,E2 -9287.043} C_VEL
LIN {X 0,Y 431.645,Z 191.863,A -85,B 0,C 180,E1 -9289.992,E2 -9289.992} C_VEL
LIN {X 0,Y 431.767,Z 187.597,A -85,B 0,C 180,E1 -9292.993,E2 -9292.993} C_VEL
LIN {X 0,Y 431.916,Z 183.388,A -85,B 0,C 180,E1 -9296.059,E2 -9296.059} C_VEL
LIN {X 0,Y 432.06,Z 179.153,A -85,B 0,C 180,E1 -9299.205,E2 -9299.205} C_VEL
LIN {X 0,Y 432.175,Z 174.887,A -85,B 0,C 180,E1 -9302.452,E2 -9302.452} C_VEL
LIN {X 0,Y 432.186,Z 173.657,A -85,B 0,C 180,E1 -9303.562,E2 -9303.562} C_VEL
LIN {X 0,Y 432.314,Z 173.635,A -85,B 0,C 180,E1 -9305.816,E2 -9305.816} C_VEL
LIN {X 0,Y 432.309,Z 173.636,A -85,B 0,C 180,E1 -9309.343,E2 -9309.343} C_VEL
LIN {X 0,Y 432.32,Z 173.634,A -85,B 0,C 180,E1 -9311.794,E2 -9311.794} C_VEL
LIN {X 0,Y 432.362,Z 173.628,A -85,B 0,C 180,E1 -9315.656,E2 -9315.656} C_VEL
LIN {X 0,Y 432.354,Z 173.626,A -85,B 0,C 180,E1 -9318.389,E2 -9318.389} C_VEL
LIN {X 0,Y 432.322,Z 173.632,A -85,B 0,C 180,E1 -9321.848,E2 -9321.848} C_VEL
LIN {X 0,Y 432.316,Z 173.635,A -85,B 0,C 180,E1 -9325.32,E2 -9325.32} C_VEL
LIN {X 0,Y 432.298,Z 173.637,A -85,B 0,C 180,E1 -9328.652,E2 -9328.652} C_VEL
LIN {X 0,Y 432.354,Z 173.628,A -85,B 0,C 180,E1 -9331.367,E2 -9331.367} C_VEL
LIN {X 0,Y 432.341,Z 173.629,A -85,B 0,C 180,E1 -9333.966,E2 -9333.966} C_VEL
LIN {X 0,Y 432.305,Z 173.634,A -85,B 0,C 180,E1 -9337.035,E2 -9337.035} C_VEL
LIN {X 0,Y 432.351,Z 173.631,A -85,B 0,C 180,E1 -9340.04,E2 -9340.04} C_VEL
LIN {X 0,Y 432.39,Z 173.624,A -85,B 0,C 180,E1 -9343.515,E2 -9343.515} C_VEL
LIN {X 0,Y 432.406,Z 173.622,A -85,B 0,C 180,E1 -9346.847,E2 -9346.847} C_VEL
LIN {X 0,Y 432.421,Z 173.62,A -85,B 0,C 180,E1 -9349.701,E2 -9349.701} C_VEL
LIN {X 0,Y 432.529,Z 173.606,A -85,B 0,C 180,E1 -9352.531,E2 -9352.531} C_VEL
LIN {X 0,Y 432.578,Z 173.6,A -85,B 0,C 180,E1 -9354.406,E2 -9354.406} C_VEL
LIN {X 0,Y 432.568,Z 173.603,A -85,B 0,C 180,E1 -9358.138,E2 -9358.138} C_VEL
LIN {X 0,Y 432.694,Z 173.588,A -85,B 0,C 180,E1 -9360,E2 -9360} C_VEL
LIN {X 0,Y 432.581,Z 173.6,A -85,B 0,C 180,E1 -9362.794,E2 -9362.794} C_VEL
LIN {X 0,Y 432.548,Z 173.603,A -85,B 0,C 180,E1 -9366.531,E2 -9366.531} C_VEL
LIN {X 0,Y 432.468,Z 173.617,A -85,B 0,C 180,E1 -9369.352,E2 -9369.352} C_VEL
LIN {X 0,Y 432.412,Z 173.621,A -85,B 0,C 180,E1 -9372.813,E2 -9372.813} C_VEL
LIN {X 0,Y 432.379,Z 173.625,A -85,B 0,C 180,E1 -9376.48,E2 -9376.48} C_VEL
LIN {X 0,Y 432.35,Z 173.629,A -85,B 0,C 180,E1 -9379.96,E2 -9379.96} C_VEL
LIN {X 0,Y 432.304,Z 173.637,A -85,B 0,C 180,E1 -9382.965,E2 -9382.965} C_VEL
LIN {X 0,Y 432.339,Z 173.628,A -85,B 0,C 180,E1 -9386.034,E2 -9386.034} C_VEL
LIN {X 0,Y 432.324,Z 173.632,A -85,B 0,C 180,E1 -9389.189,E2 -9389.189} C_VEL
LIN {X 0,Y 432.298,Z 173.637,A -85,B 0,C 180,E1 -9392.295,E2 -9392.295} C_VEL
LIN {X 0,Y 432.315,Z 173.635,A -85,B 0,C 180,E1 -9394.679,E2 -9394.679} C_VEL
LIN {X 0,Y 432.329,Z 173.633,A -85,B 0,C 180,E1 -9398.151,E2 -9398.151} C_VEL
LIN {X 0,Y 432.352,Z 173.628,A -85,B 0,C 180,E1 -9401.61,E2 -9401.61} C_VEL
LIN {X 0,Y 432.36,Z 173.632,A -85,B 0,C 180,E1 -9404.344,E2 -9404.344} C_VEL
LIN {X 0,Y 432.347,Z 173.633,A -85,B 0,C 180,E1 -9407.012,E2 -9407.012} C_VEL
LIN {X 0,Y 432.41,Z 173.742,A -85,B 0,C 180,E1 -9410.215,E2 -9410.215} C_VEL
LIN {X 0,Y 433.212,Z 178.908,A -85,B 0,C 180,E1 -9413.116,E2 -9413.116} C_VEL
LIN {X 0,Y 433.41,Z 182.186,A -85,B 0,C 180,E1 -9414.858,E2 -9414.858} C_VEL
LIN {X 0,Y 433.028,Z 188.735,A -85,B 0,C 180,E1 -9418.169,E2 -9418.169} C_VEL
LIN {X 0,Y 432.621,Z 195.2,A -85,B 0,C 180,E1 -9421.311,E2 -9421.311} C_VEL
LIN {X 0,Y 432.326,Z 201.899,A -85,B 0,C 180,E1 -9424.485,E2 -9424.485} C_VEL
LIN {X 0,Y 432.011,Z 209.564,A -85,B 0,C 180,E1 -9428.03,E2 -9428.03} C_VEL
LIN {X 0,Y 431.695,Z 217.176,A -85,B 0,C 180,E1 -9431.493,E2 -9431.493} C_VEL
LIN {X 0,Y 431.569,Z 221.579,A -85,B 0,C 180,E1 -9433.407,E2 -9433.407} C_VEL
LIN {X 0,Y 433.74,Z 234.713,A -85,B 0,C 180,E1 -9433.867,E2 -9433.867} C_VEL
LIN {X 0,Y 435.329,Z 246.357,A -85,B 0,C 180,E1 -9434.433,E2 -9434.433} C_VEL
LIN {X 0,Y 434.725,Z 258.448,A -85,B 0,C 180,E1 -9435.131,E2 -9435.131} C_VEL
LIN {X 0,Y 434.039,Z 270.521,A -85,B 0,C 180,E1 -9436.04,E2 -9436.04} C_VEL
LIN {X 0,Y 433.496,Z 280.563,A -85,B 0,C 180,E1 -9437.002,E2 -9437.002} C_VEL
LIN {X 0,Y 432.928,Z 289.596,A -85,B 0,C 180,E1 -9438.056,E2 -9438.056} C_VEL
LIN {X 0,Y 432.262,Z 299.376,A -85,B 0,C 180,E1 -9439.462,E2 -9439.462} C_VEL
LIN {X 0,Y 431.838,Z 307.201,A -85,B 0,C 180,E1 -9440.871,E2 -9440.871} C_VEL
LIN {X 0,Y 431.492,Z 314.372,A -85,B 0,C 180,E1 -9442.514,E2 -9442.514} C_VEL
LIN {X 0,Y 431.283,Z 319.462,A -85,B 0,C 180,E1 -9444.021,E2 -9444.021} C_VEL
LIN {X 0,Y 431.27,Z 322.824,A -85,B 0,C 180,E1 -9445.327,E2 -9445.327} C_VEL
LIN {X 0,Y 431.187,Z 324.717,A -85,B 0,C 180,E1 -9446.263,E2 -9446.263} C_VEL
LIN {X 0,Y 431.235,Z 326.155,A -85,B 0,C 180,E1 -9447.198,E2 -9447.198} C_VEL
LIN {X 0,Y 431.202,Z 327.173,A -85,B 0,C 180,E1 -9448.133,E2 -9448.133} C_VEL
LIN {X 0,Y 431.168,Z 328.046,A -85,B 0,C 180,E1 -9450.001,E2 -9450.001} C_VEL
LIN {X 0,Y 431.169,Z 327.867,A -85,B 0,C 180,E1 -9450.935,E2 -9450.935} C_VEL
LIN {X 0,Y 431.203,Z 327.282,A -85,B 0,C 180,E1 -9451.869,E2 -9451.869} C_VEL
LIN {X 0,Y 431.235,Z 326.31,A -85,B 0,C 180,E1 -9452.803,E2 -9452.803} C_VEL
LIN {X 0,Y 431.186,Z 324.94,A -85,B 0,C 180,E1 -9453.739,E2 -9453.739} C_VEL
LIN {X 0,Y 431.294,Z 322.05,A -85,B 0,C 180,E1 -9455.142,E2 -9455.142} C_VEL
LIN {X 0,Y 431.377,Z 318.131,A -85,B 0,C 180,E1 -9456.549,E2 -9456.549} C_VEL
LIN {X 0,Y 431.586,Z 313.086,A -85,B 0,C 180,E1 -9457.956,E2 -9457.956} C_VEL
LIN {X 0,Y 431.949,Z 306.752,A -85,B 0,C 180,E1 -9459.364,E2 -9459.364} C_VEL
LIN {X 0,Y 432.394,Z 298.824,A -85,B 0,C 180,E1 -9460.773,E2 -9460.773} C_VEL
LIN {X 0,Y 433.058,Z 290.759,A -85,B 0,C 180,E1 -9461.941,E2 -9461.941} C_VEL
LIN {X 0,Y 433.639,Z 280.926,A -85,B 0,C 180,E1 -9463.114,E2 -9463.114} C_VEL
LIN {X 0,Y 434.219,Z 271.286,A -85,B 0,C 180,E1 -9464.05,E2 -9464.05} C_VEL
LIN {X 0,Y 434.892,Z 260.915,A -85,B 0,C 180,E1 -9464.865,E2 -9464.865} C_VEL
LIN {X 0,Y 435.593,Z 248.475,A -85,B 0,C 180,E1 -9465.619,E2 -9465.619} C_VEL
LIN {X 0,Y 434.548,Z 237.906,A -85,B 0,C 180,E1 -9466.16,E2 -9466.16} C_VEL
LIN {X 0,Y 432.272,Z 225.083,A -85,B 0,C 180,E1 -9466.678,E2 -9466.678} C_VEL
LIN {X 0,Y 431.606,Z 221.24,A -85,B 0,C 180,E1 -9466.829,E2 -9466.829} C_VEL
LIN {X 0,Y 431.858,Z 213.246,A -85,B 0,C 180,E1 -9470.48,E2 -9470.48} C_VEL
LIN {X 0,Y 432.141,Z 206.807,A -85,B 0,C 180,E1 -9473.48,E2 -9473.48} C_VEL
LIN {X 0,Y 432.491,Z 200.062,A -85,B 0,C 180,E1 -9476.651,E2 -9476.651} C_VEL
LIN {X 0,Y 432.954,Z 192.715,A -85,B 0,C 180,E1 -9480.211,E2 -9480.211} C_VEL
LIN {X 0,Y 433.317,Z 186.261,A -85,B 0,C 180,E1 -9483.464,E2 -9483.464} C_VEL
LIN {X 0,Y 433.52,Z 181.724,A -85,B 0,C 180,E1 -9485.848,E2 -9485.848} C_VEL
LIN {X 0,Y 433.046,Z 177.717,A -85,B 0,C 180,E1 -9488.074,E2 -9488.074} C_VEL
LIN {X 0,Y 432.34,Z 173.633,A -85,B 0,C 180,E1 -9490.556,E2 -9490.556} C_VEL
LIN {X 0,Y 432.354,Z 173.628,A -85,B 0,C 180,E1 -9493.053,E2 -9493.053} C_VEL
LIN {X 0,Y 432.321,Z 173.635,A -85,B 0,C 180,E1 -9495.663,E2 -9495.663} C_VEL
LIN {X 0,Y 432.318,Z 173.633,A -85,B 0,C 180,E1 -9498.397,E2 -9498.397} C_VEL
LIN {X 0,Y 432.317,Z 173.635,A -85,B 0,C 180,E1 -9501.848,E2 -9501.848} C_VEL
LIN {X 0,Y 432.323,Z 173.636,A -85,B 0,C 180,E1 -9505.321,E2 -9505.321} C_VEL
LIN {X 0,Y 432.302,Z 173.635,A -85,B 0,C 180,E1 -9508.652,E2 -9508.652} C_VEL
LIN {X 0,Y 432.361,Z 173.628,A -85,B 0,C 180,E1 -9511.875,E2 -9511.875} C_VEL
LIN {X 0,Y 432.332,Z 173.634,A -85,B 0,C 180,E1 -9514.998,E2 -9514.998} C_VEL
LIN {X 0,Y 432.365,Z 173.625,A -85,B 0,C 180,E1 -9518.046,E2 -9518.046} C_VEL
LIN {X 0,Y 432.365,Z 173.629,A -85,B 0,C 180,E1 -9521.029,E2 -9521.029} C_VEL
LIN {X 0,Y 432.418,Z 173.62,A -85,B 0,C 180,E1 -9523.961,E2 -9523.961} C_VEL
LIN {X 0,Y 432.457,Z 173.615,A -85,B 0,C 180,E1 -9527.804,E2 -9527.804} C_VEL
LIN {X 0,Y 432.469,Z 173.612,A -85,B 0,C 180,E1 -9531.59,E2 -9531.59} C_VEL
LIN {X 0,Y 432.587,Z 173.602,A -85,B 0,C 180,E1 -9534.406,E2 -9534.406} C_VEL
LIN {X 0,Y 432.575,Z 173.603,A -85,B 0,C 180,E1 -9538.138,E2 -9538.138} C_VEL
LIN {X 0,Y 432.701,Z 173.587,A -85,B 0,C 180,E1 -9540,E2 -9540} C_VEL
LIN {X 0,Y 432.59,Z 173.598,A -85,B 0,C 180,E1 -9542.794,E2 -9542.794} C_VEL
LIN {X 0,Y 432.55,Z 173.605,A -85,B 0,C 180,E1 -9546.531,E2 -9546.531} C_VEL
LIN {X 0,Y 432.417,Z 173.621,A -85,B 0,C 180,E1 -9549.354,E2 -9549.354} C_VEL
LIN {X 0,Y 432.406,Z 173.621,A -85,B 0,C 180,E1 -9552.804,E2 -9552.804} C_VEL
LIN {X 0,Y 432.421,Z 173.618,A -85,B 0,C 180,E1 -9556.494,E2 -9556.494} C_VEL
LIN {X 0,Y 432.317,Z 173.634,A -85,B 0,C 180,E1 -9559.962,E2 -9559.962} C_VEL
LIN {X 0,Y 432.298,Z 173.637,A -85,B 0,C 180,E1 -9562.966,E2 -9562.966} C_VEL
LIN {X 0,Y 432.344,Z 173.629,A -85,B 0,C 180,E1 -9566.034,E2 -9566.034} C_VEL
LIN {X 0,Y 432.333,Z 173.634,A -85,B 0,C 180,E1 -9569.189,E2 -9569.189} C_VEL
LIN {X 0,Y 432.308,Z 173.633,A -85,B 0,C 180,E1 -9572.295,E2 -9572.295} C_VEL
LIN {X 0,Y 432.324,Z 173.634,A -85,B 0,C 180,E1 -9574.679,E2 -9574.679} C_VEL
LIN {X 0,Y 432.321,Z 173.632,A -85,B 0,C 180,E1 -9578.152,E2 -9578.152} C_VEL
LIN {X 0,Y 432.32,Z 173.631,A -85,B 0,C 180,E1 -9581.604,E2 -9581.604} C_VEL
LIN {X 0,Y 432.324,Z 173.633,A -85,B 0,C 180,E1 -9584.349,E2 -9584.349} C_VEL
LIN {X 0,Y 432.311,Z 173.636,A -85,B 0,C 180,E1 -9587.018,E2 -9587.018} C_VEL
LIN {X 0,Y 432.307,Z 173.634,A -85,B 0,C 180,E1 -9589.826,E2 -9589.826} C_VEL
LIN {X 0,Y 432.26,Z 173.643,A -85,B 0,C 180,E1 -9591.845,E2 -9591.845} C_VEL
LIN {X 0,Y 432.24,Z 174.788,A -85,B 0,C 180,E1 -9593.018,E2 -9593.018} C_VEL
LIN {X 0,Y 432.199,Z 178.62,A -85,B 0,C 180,E1 -9596.029,E2 -9596.029} C_VEL
LIN {X 0,Y 431.998,Z 183.272,A -85,B 0,C 180,E1 -9599.57,E2 -9599.57} C_VEL
LIN {X 0,Y 431.798,Z 187.771,A -85,B 0,C 180,E1 -9602.889,E2 -9602.889} C_VEL
LIN {X 0,Y 431.726,Z 192.116,A -85,B 0,C 180,E1 -9605.986,E2 -9605.986} C_VEL
LIN {X 0,Y 431.549,Z 196.485,A -85,B 0,C 180,E1 -9609.006,E2 -9609.006} C_VEL
LIN {X 0,Y 431.544,Z 199.951,A -85,B 0,C 180,E1 -9611.277,E2 -9611.277} C_VEL
LIN {X 0,Y 434.635,Z 213.359,A -85,B 0,C 180,E1 -9611.832,E2 -9611.832} C_VEL
LIN {X 0,Y 436.048,Z 221.744,A -85,B 0,C 180,E1 -9612.261,E2 -9612.261} C_VEL
LIN {X 0,Y 435.551,Z 233.911,A -85,B 0,C 180,E1 -9612.953,E2 -9612.953} C_VEL
LIN {X 0,Y 434.834,Z 245.536,A -85,B 0,C 180,E1 -9613.812,E2 -9613.812} C_VEL
LIN {X 0,Y 434.17,Z 255.623,A -85,B 0,C 180,E1 -9614.75,E2 -9614.75} C_VEL
LIN {X 0,Y 433.516,Z 265.779,A -85,B 0,C 180,E1 -9615.926,E2 -9615.926} C_VEL
LIN {X 0,Y 432.904,Z 274.005,A -85,B 0,C 180,E1 -9617.095,E2 -9617.095} C_VEL
LIN {X 0,Y 432.487,Z 282.13,A -85,B 0,C 180,E1 -9618.518,E2 -9618.518} C_VEL
LIN {X 0,Y 432.001,Z 287.619,A -85,B 0,C 180,E1 -9619.691,E2 -9619.691} C_VEL
LIN {X 0,Y 431.728,Z 292.975,A -85,B 0,C 180,E1 -9621.104,E2 -9621.104} C_VEL
LIN {X 0,Y 431.489,Z 297.154,A -85,B 0,C 180,E1 -9622.513,E2 -9622.513} C_VEL
LIN {X 0,Y 431.373,Z 299.729,A -85,B 0,C 180,E1 -9623.632,E2 -9623.632} C_VEL
LIN {X 0,Y 431.249,Z 302.424,A -85,B 0,C 180,E1 -9625.326,E2 -9625.326} C_VEL
LIN {X 0,Y 431.274,Z 303.891,A -85,B 0,C 180,E1 -9627.197,E2 -9627.197} C_VEL
LIN {X 0,Y 431.198,Z 303.937,A -85,B 0,C 180,E1 -9628.371,E2 -9628.371} C_VEL
LIN {X 0,Y 430.488,Z 303.727,A -85,B 0,C 180,E1 -9629.15,E2 -9629.15} C_VEL
LIN {X 0,Y 427.624,Z 302.782,A -85,B 0,C 180,E1 -9630.412,E2 -9630.412} C_VEL
LIN {X 0,Y 425.273,Z 301.528,A -85,B 0,C 180,E1 -9631.422,E2 -9631.422} C_VEL
LIN {X 0,Y 424.329,Z 300.246,A -85,B 0,C 180,E1 -9632.193,E2 -9632.193} C_VEL
LIN {X 0,Y 424.286,Z 299.695,A -85,B 0,C 180,E1 -9632.451,E2 -9632.451} C_VEL
LIN {X 0,Y 424.531,Z 296.587,A -85,B 0,C 180,E1 -9633.796,E2 -9633.796} C_VEL
LIN {X 0,Y 424.672,Z 292.206,A -85,B 0,C 180,E1 -9635.221,E2 -9635.221} C_VEL
LIN {X 0,Y 425.031,Z 286.634,A -85,B 0,C 180,E1 -9636.646,E2 -9636.646} C_VEL
LIN {X 0,Y 425.431,Z 279.669,A -85,B 0,C 180,E1 -9638.071,E2 -9638.071} C_VEL
LIN {X 0,Y 426.072,Z 270.95,A -85,B 0,C 180,E1 -9639.493,E2 -9639.493} C_VEL
LIN {X 0,Y 426.798,Z 261.05,A -85,B 0,C 180,E1 -9640.794,E2 -9640.794} C_VEL
LIN {X 0,Y 427.389,Z 250.949,A -85,B 0,C 180,E1 -9641.86,E2 -9641.86} C_VEL
LIN {X 0,Y 427.85,Z 242.833,A -85,B 0,C 180,E1 -9642.569,E2 -9642.569} C_VEL
LIN {X 0,Y 428.441,Z 231.068,A -85,B 0,C 180,E1 -9643.397,E2 -9643.397} C_VEL
LIN {X 0,Y 428.755,Z 221.108,A -85,B 0,C 180,E1 -9643.946,E2 -9643.946} C_VEL
LIN {X 0,Y 426.179,Z 207.956,A -85,B 0,C 180,E1 -9644.583,E2 -9644.583} C_VEL
LIN {X 0,Y 424.445,Z 199.938,A -85,B 0,C 180,E1 -9644.9,E2 -9644.9} C_VEL
LIN {X 0,Y 424.522,Z 196.386,A -85,B 0,C 180,E1 -9647.335,E2 -9647.335} C_VEL
LIN {X 0,Y 424.606,Z 192.066,A -85,B 0,C 180,E1 -9650.338,E2 -9650.338} C_VEL
LIN {X 0,Y 424.735,Z 187.774,A -85,B 0,C 180,E1 -9653.396,E2 -9653.396} C_VEL
LIN {X 0,Y 424.894,Z 183.286,A -85,B 0,C 180,E1 -9656.722,E2 -9656.722} C_VEL
LIN {X 0,Y 425.018,Z 179.307,A -85,B 0,C 180,E1 -9659.737,E2 -9659.737} C_VEL
LIN {X 0,Y 425.121,Z 175.03,A -85,B 0,C 180,E1 -9663.059,E2 -9663.059} C_VEL
LIN {X 0,Y 425.21,Z 174.522,A -85,B 0,C 180,E1 -9664.267,E2 -9664.267} C_VEL
LIN {X 0,Y 425.264,Z 174.513,A -85,B 0,C 180,E1 -9667.508,E2 -9667.508} C_VEL
LIN {X 0,Y 425.266,Z 174.511,A -85,B 0,C 180,E1 -9670.517,E2 -9670.517} C_VEL
LIN {X 0,Y 425.249,Z 174.516,A -85,B 0,C 180,E1 -9673.349,E2 -9673.349} C_VEL
LIN {X 0,Y 425.299,Z 174.506,A -85,B 0,C 180,E1 -9676.638,E2 -9676.638} C_VEL
LIN {X 0,Y 425.29,Z 174.507,A -85,B 0,C 180,E1 -9679.873,E2 -9679.873} C_VEL
LIN {X 0,Y 425.258,Z 174.513,A -85,B 0,C 180,E1 -9682.486,E2 -9682.486} C_VEL
LIN {X 0,Y 425.283,Z 174.509,A -85,B 0,C 180,E1 -9685.815,E2 -9685.815} C_VEL
LIN {X 0,Y 425.274,Z 174.512,A -85,B 0,C 180,E1 -9689.234,E2 -9689.234} C_VEL
LIN {X 0,Y 425.324,Z 174.505,A -85,B 0,C 180,E1 -9692.44,E2 -9692.44} C_VEL
LIN {X 0,Y 425.329,Z 174.501,A -85,B 0,C 180,E1 -9695.6,E2 -9695.6} C_VEL
LIN {X 0,Y 425.29,Z 174.51,A -85,B 0,C 180,E1 -9698.681,E2 -9698.681} C_VEL
LIN {X 0,Y 425.301,Z 174.507,A -85,B 0,C 180,E1 -9701.701,E2 -9701.701} C_VEL
LIN {X 0,Y 425.341,Z 174.504,A -85,B 0,C 180,E1 -9704.67,E2 -9704.67} C_VEL
LIN {X 0,Y 425.406,Z 174.495,A -85,B 0,C 180,E1 -9707.598,E2 -9707.598} C_VEL
LIN {X 0,Y 425.444,Z 174.488,A -85,B 0,C 180,E1 -9711.45,E2 -9711.45} C_VEL
LIN {X 0,Y 425.555,Z 174.476,A -85,B 0,C 180,E1 -9714.313,E2 -9714.313} C_VEL
LIN {X 0,Y 425.538,Z 174.479,A -85,B 0,C 180,E1 -9718.107,E2 -9718.107} C_VEL
LIN {X 0,Y 425.664,Z 174.463,A -85,B 0,C 180,E1 -9720,E2 -9720} C_VEL
LIN {X 0,Y 425.533,Z 174.478,A -85,B 0,C 180,E1 -9722.84,E2 -9722.84} C_VEL
LIN {X 0,Y 425.55,Z 174.479,A -85,B 0,C 180,E1 -9725.687,E2 -9725.687} C_VEL
LIN {X 0,Y 425.442,Z 174.487,A -85,B 0,C 180,E1 -9728.55,E2 -9728.55} C_VEL
LIN {X 0,Y 425.4,Z 174.493,A -85,B 0,C 180,E1 -9732.402,E2 -9732.402} C_VEL
LIN {X 0,Y 425.355,Z 174.5,A -85,B 0,C 180,E1 -9736.313,E2 -9736.313} C_VEL
LIN {X 0,Y 425.33,Z 174.505,A -85,B 0,C 180,E1 -9739.649,E2 -9739.649} C_VEL
LIN {X 0,Y 425.288,Z 174.51,A -85,B 0,C 180,E1 -9743.366,E2 -9743.366} C_VEL
LIN {X 0,Y 425.32,Z 174.508,A -85,B 0,C 180,E1 -9746.846,E2 -9746.846} C_VEL
LIN {X 0,Y 425.29,Z 174.507,A -85,B 0,C 180,E1 -9749.72,E2 -9749.72} C_VEL
LIN {X 0,Y 425.256,Z 174.514,A -85,B 0,C 180,E1 -9753.05,E2 -9753.05} C_VEL
LIN {X 0,Y 425.26,Z 174.513,A -85,B 0,C 180,E1 -9755.931,E2 -9755.931} C_VEL
LIN {X 0,Y 425.29,Z 174.509,A -85,B 0,C 180,E1 -9759.048,E2 -9759.048} C_VEL
LIN {X 0,Y 425.312,Z 174.508,A -85,B 0,C 180,E1 -9762.649,E2 -9762.649} C_VEL
LIN {X 0,Y 425.317,Z 174.508,A -85,B 0,C 180,E1 -9766.056,E2 -9766.056} C_VEL
LIN {X 0,Y 425.274,Z 174.517,A -85,B 0,C 180,E1 -9769.481,E2 -9769.481} C_VEL
LIN {X 0,Y 425.363,Z 174.674,A -85,B 0,C 180,E1 -9770.022,E2 -9770.022} C_VEL
LIN {X 0,Y 426.173,Z 179.852,A -85,B 0,C 180,E1 -9772.996,E2 -9772.996} C_VEL
LIN {X 0,Y 426.389,Z 183.132,A -85,B 0,C 180,E1 -9774.772,E2 -9774.772} C_VEL
LIN {X 0,Y 426.012,Z 189.679,A -85,B 0,C 180,E1 -9778.139,E2 -9778.139} C_VEL
LIN {X 0,Y 425.619,Z 195.582,A -85,B 0,C 180,E1 -9781.064,E2 -9781.064} C_VEL
LIN {X 0,Y 425.27,Z 202.819,A -85,B 0,C 180,E1 -9784.556,E2 -9784.556} C_VEL
LIN {X 0,Y 424.935,Z 209.802,A -85,B 0,C 180,E1 -9787.848,E2 -9787.848} C_VEL
LIN {X 0,Y 424.648,Z 216.967,A -85,B 0,C 180,E1 -9791.174,E2 -9791.174} C_VEL
LIN {X 0,Y 424.5,Z 221.195,A -85,B 0,C 180,E1 -9793.13,E2 -9793.13} C_VEL
LIN {X 0,Y 426.771,Z 234.508,A -85,B 0,C 180,E1 -9793.609,E2 -9793.609} C_VEL
LIN {X 0,Y 428.398,Z 247.058,A -85,B 0,C 180,E1 -9794.236,E2 -9794.236} C_VEL
LIN {X 0,Y 427.766,Z 259.842,A -85,B 0,C 180,E1 -9795.005,E2 -9795.005} C_VEL
LIN {X 0,Y 427.018,Z 271.745,A -85,B 0,C 180,E1 -9795.951,E2 -9795.951} C_VEL
LIN {X 0,Y 426.386,Z 282.404,A -85,B 0,C 180,E1 -9797.024,E2 -9797.024} C_VEL
LIN {X 0,Y 425.827,Z 291.097,A -85,B 0,C 180,E1 -9798.096,E2 -9798.096} C_VEL
LIN {X 0,Y 425.254,Z 299.102,A -85,B 0,C 180,E1 -9799.286,E2 -9799.286} C_VEL
LIN {X 0,Y 424.798,Z 306.946,A -85,B 0,C 180,E1 -9800.719,E2 -9800.719} C_VEL
LIN {X 0,Y 424.52,Z 312.283,A -85,B 0,C 180,E1 -9801.912,E2 -9801.912} C_VEL
LIN {X 0,Y 424.27,Z 318.465,A -85,B 0,C 180,E1 -9803.667,E2 -9803.667} C_VEL
LIN {X 0,Y 424.199,Z 322.6,A -85,B 0,C 180,E1 -9805.249,E2 -9805.249} C_VEL
LIN {X 0,Y 424.098,Z 324.497,A -85,B 0,C 180,E1 -9806.2,E2 -9806.2} C_VEL
LIN {X 0,Y 424.131,Z 325.943,A -85,B 0,C 180,E1 -9807.151,E2 -9807.151} C_VEL
LIN {X 0,Y 424.128,Z 326.966,A -85,B 0,C 180,E1 -9808.102,E2 -9808.102} C_VEL
LIN {X 0,Y 424.085,Z 327.847,A -85,B 0,C 180,E1 -9810.001,E2 -9810.001} C_VEL
LIN {X 0,Y 424.088,Z 327.676,A -85,B 0,C 180,E1 -9810.95,E2 -9810.95} C_VEL
LIN {X 0,Y 424.129,Z 327.095,A -85,B 0,C 180,E1 -9811.9,E2 -9811.9} C_VEL
LIN {X 0,Y 424.131,Z 326.125,A -85,B 0,C 180,E1 -9812.85,E2 -9812.85} C_VEL
LIN {X 0,Y 424.098,Z 324.76,A -85,B 0,C 180,E1 -9813.801,E2 -9813.801} C_VEL
LIN {X 0,Y 424.206,Z 321.878,A -85,B 0,C 180,E1 -9815.228,E2 -9815.228} C_VEL
LIN {X 0,Y 424.302,Z 317.968,A -85,B 0,C 180,E1 -9816.658,E2 -9816.658} C_VEL
LIN {X 0,Y 424.53,Z 312.932,A -85,B 0,C 180,E1 -9818.089,E2 -9818.089} C_VEL
LIN {X 0,Y 424.9,Z 306.612,A -85,B 0,C 180,E1 -9819.521,E2 -9819.521} C_VEL
LIN {X 0,Y 425.404,Z 298.7,A -85,B 0,C 180,E1 -9820.952,E2 -9820.952} C_VEL
LIN {X 0,Y 426.084,Z 290.651,A -85,B 0,C 180,E1 -9822.14,E2 -9822.14} C_VEL
LIN {X 0,Y 426.693,Z 280.837,A -85,B 0,C 180,E1 -9823.332,E2 -9823.332} C_VEL
LIN {X 0,Y 427.43,Z 269.889,A -85,B 0,C 180,E1 -9824.4,E2 -9824.4} C_VEL
LIN {X 0,Y 428.115,Z 259.165,A -85,B 0,C 180,E1 -9825.227,E2 -9825.227} C_VEL
LIN {X 0,Y 428.704,Z 247.381,A -85,B 0,C 180,E1 -9825.937,E2 -9825.937} C_VEL
LIN {X 0,Y 427.045,Z 234.388,A -85,B 0,C 180,E1 -9826.599,E2 -9826.599} C_VEL
LIN {X 0,Y 424.531,Z 221.107,A -85,B 0,C 180,E1 -9827.105,E2 -9827.105} C_VEL
LIN {X 0,Y 424.773,Z 214.173,A -85,B 0,C 180,E1 -9830.331,E2 -9830.331} C_VEL
LIN {X 0,Y 425.083,Z 207.743,A -85,B 0,C 180,E1 -9833.377,E2 -9833.377} C_VEL
LIN {X 0,Y 425.406,Z 201.268,A -85,B 0,C 180,E1 -9836.49,E2 -9836.49} C_VEL
LIN {X 0,Y 425.907,Z 194.772,A -85,B 0,C 180,E1 -9839.671,E2 -9839.671} C_VEL
LIN {X 0,Y 426.223,Z 188.324,A -85,B 0,C 180,E1 -9842.964,E2 -9842.964} C_VEL
LIN {X 0,Y 426.534,Z 184.057,A -85,B 0,C 180,E1 -9845.216,E2 -9845.216} C_VEL
LIN {X 0,Y 426.166,Z 179.663,A -85,B 0,C 180,E1 -9847.667,E2 -9847.667} C_VEL
LIN {X 0,Y 425.287,Z 174.51,A -85,B 0,C 180,E1 -9850.796,E2 -9850.796} C_VEL
LIN {X 0,Y 425.323,Z 174.506,A -85,B 0,C 180,E1 -9853.945,E2 -9853.945} C_VEL
LIN {X 0,Y 425.261,Z 174.515,A -85,B 0,C 180,E1 -9857.345,E2 -9857.345} C_VEL
LIN {X 0,Y 425.27,Z 174.513,A -85,B 0,C 180,E1 -9859.871,E2 -9859.871} C_VEL
LIN {X 0,Y 425.261,Z 174.511,A -85,B 0,C 180,E1 -9862.487,E2 -9862.487} C_VEL
LIN {X 0,Y 425.29,Z 174.508,A -85,B 0,C 180,E1 -9865.816,E2 -9865.816} C_VEL
LIN {X 0,Y 425.272,Z 174.513,A -85,B 0,C 180,E1 -9869.238,E2 -9869.238} C_VEL
LIN {X 0,Y 425.328,Z 174.504,A -85,B 0,C 180,E1 -9872.441,E2 -9872.441} C_VEL
LIN {X 0,Y 425.332,Z 174.503,A -85,B 0,C 180,E1 -9875.601,E2 -9875.601} C_VEL
LIN {X 0,Y 425.298,Z 174.509,A -85,B 0,C 180,E1 -9878.682,E2 -9878.682} C_VEL
LIN {X 0,Y 425.313,Z 174.504,A -85,B 0,C 180,E1 -9881.702,E2 -9881.702} C_VEL
LIN {X 0,Y 425.33,Z 174.506,A -85,B 0,C 180,E1 -9884.67,E2 -9884.67} C_VEL
LIN {X 0,Y 425.406,Z 174.493,A -85,B 0,C 180,E1 -9887.598,E2 -9887.598} C_VEL
LIN {X 0,Y 425.42,Z 174.49,A -85,B 0,C 180,E1 -9891.45,E2 -9891.45} C_VEL
LIN {X 0,Y 425.564,Z 174.477,A -85,B 0,C 180,E1 -9894.314,E2 -9894.314} C_VEL
LIN {X 0,Y 425.545,Z 174.479,A -85,B 0,C 180,E1 -9898.107,E2 -9898.107} C_VEL
LIN {X 0,Y 425.671,Z 174.463,A -85,B 0,C 180,E1 -9900,E2 -9900} C_VEL
LIN {X 0,Y 425.542,Z 174.475,A -85,B 0,C 180,E1 -9902.84,E2 -9902.84} C_VEL
LIN {X 0,Y 425.554,Z 174.477,A -85,B 0,C 180,E1 -9905.687,E2 -9905.687} C_VEL
LIN {X 0,Y 425.417,Z 174.493,A -85,B 0,C 180,E1 -9908.551,E2 -9908.551} C_VEL
LIN {X 0,Y 425.387,Z 174.496,A -85,B 0,C 180,E1 -9912.403,E2 -9912.403} C_VEL
LIN {X 0,Y 425.389,Z 174.494,A -85,B 0,C 180,E1 -9916.312,E2 -9916.312} C_VEL
LIN {X 0,Y 425.307,Z 174.509,A -85,B 0,C 180,E1 -9919.637,E2 -9919.637} C_VEL
LIN {X 0,Y 425.286,Z 174.511,A -85,B 0,C 180,E1 -9923.367,E2 -9923.367} C_VEL
LIN {X 0,Y 425.328,Z 174.504,A -85,B 0,C 180,E1 -9926.845,E2 -9926.845} C_VEL
LIN {X 0,Y 425.3,Z 174.507,A -85,B 0,C 180,E1 -9929.719,E2 -9929.719} C_VEL
LIN {X 0,Y 425.266,Z 174.514,A -85,B 0,C 180,E1 -9933.05,E2 -9933.05} C_VEL
LIN {X 0,Y 425.267,Z 174.51,A -85,B 0,C 180,E1 -9935.93,E2 -9935.93} C_VEL
LIN {X 0,Y 425.269,Z 174.514,A -85,B 0,C 180,E1 -9939.043,E2 -9939.043} C_VEL
LIN {X 0,Y 425.278,Z 174.508,A -85,B 0,C 180,E1 -9941.96,E2 -9941.96} C_VEL
LIN {X 0,Y 425.275,Z 174.51,A -85,B 0,C 180,E1 -9945.285,E2 -9945.285} C_VEL
LIN {X 0,Y 425.264,Z 174.514,A -85,B 0,C 180,E1 -9948.623,E2 -9948.623} C_VEL
LIN {X 0,Y 425.258,Z 174.517,A -85,B 0,C 180,E1 -9951.099,E2 -9951.099} C_VEL
LIN {X 0,Y 425.198,Z 175.111,A -85,B 0,C 180,E1 -9952.503,E2 -9952.503} C_VEL
LIN {X 0,Y 425.165,Z 179.148,A -85,B 0,C 180,E1 -9955.742,E2 -9955.742} C_VEL
LIN {X 0,Y 424.959,Z 183.778,A -85,B 0,C 180,E1 -9959.315,E2 -9959.315} C_VEL
LIN {X 0,Y 424.779,Z 187.892,A -85,B 0,C 180,E1 -9962.404,E2 -9962.404} C_VEL
LIN {X 0,Y 424.679,Z 192.26,A -85,B 0,C 180,E1 -9965.562,E2 -9965.562} C_VEL
LIN {X 0,Y 424.489,Z 196.63,A -85,B 0,C 180,E1 -9968.64,E2 -9968.64} C_VEL
LIN {X 0,Y 424.483,Z 199.995,A -85,B 0,C 180,E1 -9970.972,E2 -9970.972} C_VEL
LIN {X 0,Y 427.525,Z 213.149,A -85,B 0,C 180,E1 -9971.525,E2 -9971.525} C_VEL
LIN {X 0,Y 429.232,Z 222.816,A -85,B 0,C 180,E1 -9972.037,E2 -9972.037} C_VEL
LIN {X 0,Y 428.676,Z 235.093,A -85,B 0,C 180,E1 -9972.761,E2 -9972.761} C_VEL
LIN {X 0,Y 427.899,Z 246.913,A -85,B 0,C 180,E1 -9973.665,E2 -9973.665} C_VEL
LIN {X 0,Y 427.193,Z 257.831,A -85,B 0,C 180,E1 -9974.739,E2 -9974.739} C_VEL
LIN {X 0,Y 426.487,Z 267.603,A -85,B 0,C 180,E1 -9975.933,E2 -9975.933} C_VEL
LIN {X 0,Y 425.815,Z 276.319,A -85,B 0,C 180,E1 -9977.244,E2 -9977.244} C_VEL
LIN {X 0,Y 425.4,Z 283.431,A -85,B 0,C 180,E1 -9978.565,E2 -9978.565} C_VEL
LIN {X 0,Y 424.87,Z 289.672,A -85,B 0,C 180,E1 -9979.998,E2 -9979.998} C_VEL
LIN {X 0,Y 424.595,Z 294.63,A -85,B 0,C 180,E1 -9981.433,E2 -9981.433} C_VEL
LIN {X 0,Y 424.347,Z 298.463,A -85,B 0,C 180,E1 -9982.864,E2 -9982.864} C_VEL
LIN {X 0,Y 424.235,Z 301.272,A -85,B 0,C 180,E1 -9984.295,E2 -9984.295} C_VEL
LIN {X 0,Y 424.179,Z 302.597,A -85,B 0,C 180,E1 -9985.248,E2 -9985.248} C_VEL
LIN {X 0,Y 424.172,Z 304.08,A -85,B 0,C 180,E1 -9987.15,E2 -9987.15} C_VEL
LIN {X 0,Y 424.12,Z 304.135,A -85,B 0,C 180,E1 -9988.362,E2 -9988.362} C_VEL
LIN {X 0,Y 424.089,Z 303.295,A -85,B 0,C 180,E1 -9989.999,E2 -9989.999} C_VEL
LIN {X 0,Y 424.125,Z 302.265,A -85,B 0,C 180,E1 -9990.949,E2 -9990.949} C_VEL
LIN {X 0,Y 424.286,Z 299.695,A -85,B 0,C 180,E1 -9992.451,E2 -9992.451} C_VEL
LIN {X 0,Y 423.732,Z 298.118,A -85,B 0,C 180,E1 -9993.216,E2 -9993.216} C_VEL
LIN {X 0,Y 421.034,Z 295.041,A -85,B 0,C 180,E1 -9994.444,E2 -9994.444} C_VEL
LIN {X 0,Y 418.366,Z 291.286,A -85,B 0,C 180,E1 -9995.648,E2 -9995.648} C_VEL
LIN {X 0,Y 417.868,Z 288.549,A -85,B 0,C 180,E1 -9996.365,E2 -9996.365} C_VEL
LIN {X 0,Y 418.345,Z 281.222,A -85,B 0,C 180,E1 -9997.965,E2 -9997.965} C_VEL
LIN {X 0,Y 418.928,Z 272.903,A -85,B 0,C 180,E1 -9999.413,E2 -9999.413} C_VEL
LIN {X 0,Y 419.597,Z 264.325,A -85,B 0,C 180,E1 -10000.616,E2 -10000.616} C_VEL
LIN {X 0,Y 420.286,Z 253.767,A -85,B 0,C 180,E1 -10001.819,E2 -10001.819} C_VEL
LIN {X 0,Y 420.824,Z 244.693,A -85,B 0,C 180,E1 -10002.66,E2 -10002.66} C_VEL
LIN {X 0,Y 421.441,Z 233.483,A -85,B 0,C 180,E1 -10003.5,E2 -10003.5} C_VEL
LIN {X 0,Y 422.014,Z 223.404,A -85,B 0,C 180,E1 -10004.084,E2 -10004.084} C_VEL
LIN {X 0,Y 419.768,Z 211.123,A -85,B 0,C 180,E1 -10004.729,E2 -10004.729} C_VEL
LIN {X 0,Y 417.412,Z 200.112,A -85,B 0,C 180,E1 -10005.189,E2 -10005.189} C_VEL
LIN {X 0,Y 417.483,Z 195.158,A -85,B 0,C 180,E1 -10008.652,E2 -10008.652} C_VEL
LIN {X 0,Y 417.643,Z 190.079,A -85,B 0,C 180,E1 -10012.251,E2 -10012.251} C_VEL
LIN {X 0,Y 417.745,Z 186.551,A -85,B 0,C 180,E1 -10014.869,E2 -10014.869} C_VEL
LIN {X 0,Y 417.915,Z 182.312,A -85,B 0,C 180,E1 -10018.088,E2 -10018.088} C_VEL
LIN {X 0,Y 418.062,Z 178.036,A -85,B 0,C 180,E1 -10021.405,E2 -10021.405} C_VEL
LIN {X 0,Y 418.076,Z 175.414,A -85,B 0,C 180,E1 -10023.689,E2 -10023.689} C_VEL
LIN {X 0,Y 418.226,Z 175.388,A -85,B 0,C 180,E1 -10026.233,E2 -10026.233} C_VEL
LIN {X 0,Y 418.23,Z 175.391,A -85,B 0,C 180,E1 -10029.68,E2 -10029.68} C_VEL
LIN {X 0,Y 418.217,Z 175.388,A -85,B 0,C 180,E1 -10032.319,E2 -10032.319} C_VEL
LIN {X 0,Y 418.245,Z 175.388,A -85,B 0,C 180,E1 -10035.109,E2 -10035.109} C_VEL
LIN {X 0,Y 418.274,Z 175.381,A -85,B 0,C 180,E1 -10037.77,E2 -10037.77} C_VEL
LIN {X 0,Y 418.241,Z 175.387,A -85,B 0,C 180,E1 -10041.556,E2 -10041.556} C_VEL
LIN {X 0,Y 418.236,Z 175.389,A -85,B 0,C 180,E1 -10045.156,E2 -10045.156} C_VEL
LIN {X 0,Y 418.221,Z 175.389,A -85,B 0,C 180,E1 -10047.469,E2 -10047.469} C_VEL
LIN {X 0,Y 418.251,Z 175.389,A -85,B 0,C 180,E1 -10050.891,E2 -10050.891} C_VEL
LIN {X 0,Y 418.247,Z 175.385,A -85,B 0,C 180,E1 -10054.094,E2 -10054.094} C_VEL
LIN {X 0,Y 418.248,Z 175.384,A -85,B 0,C 180,E1 -10057.535,E2 -10057.535} C_VEL
LIN {X 0,Y 418.286,Z 175.383,A -85,B 0,C 180,E1 -10060.364,E2 -10060.364} C_VEL
LIN {X 0,Y 418.294,Z 175.379,A -85,B 0,C 180,E1 -10063.403,E2 -10063.403} C_VEL
LIN {X 0,Y 418.326,Z 175.375,A -85,B 0,C 180,E1 -10066.991,E2 -10066.991} C_VEL
LIN {X 0,Y 418.386,Z 175.37,A -85,B 0,C 180,E1 -10070.329,E2 -10070.329} C_VEL
LIN {X 0,Y 418.486,Z 175.354,A -85,B 0,C 180,E1 -10073.249,E2 -10073.249} C_VEL
LIN {X 0,Y 418.317,Z 175.376,A -85,B 0,C 180,E1 -10075.181,E2 -10075.181} C_VEL
LIN {X 0,Y 418.508,Z 175.355,A -85,B 0,C 180,E1 -10078.075,E2 -10078.075} C_VEL
LIN {X 0,Y 418.634,Z 175.339,A -85,B 0,C 180,E1 -10080,E2 -10080} C_VEL
LIN {X 0,Y 418.487,Z 175.355,A -85,B 0,C 180,E1 -10082.888,E2 -10082.888} C_VEL
LIN {X 0,Y 418.505,Z 175.357,A -85,B 0,C 180,E1 -10085.783,E2 -10085.783} C_VEL
LIN {X 0,Y 418.394,Z 175.366,A -85,B 0,C 180,E1 -10088.695,E2 -10088.695} C_VEL
LIN {X 0,Y 418.339,Z 175.373,A -85,B 0,C 180,E1 -10092.615,E2 -10092.615} C_VEL
LIN {X 0,Y 418.27,Z 175.384,A -85,B 0,C 180,E1 -10095.595,E2 -10095.595} C_VEL
LIN {X 0,Y 418.251,Z 175.386,A -85,B 0,C 180,E1 -10098.618,E2 -10098.618} C_VEL
LIN {X 0,Y 418.232,Z 175.388,A -85,B 0,C 180,E1 -10101.696,E2 -10101.696} C_VEL
LIN {X 0,Y 418.255,Z 175.387,A -85,B 0,C 180,E1 -10104.866,E2 -10104.866} C_VEL
LIN {X 0,Y 418.267,Z 175.381,A -85,B 0,C 180,E1 -10108.065,E2 -10108.065} C_VEL
LIN {X 0,Y 418.189,Z 175.393,A -85,B 0,C 180,E1 -10111.398,E2 -10111.398} C_VEL
LIN {X 0,Y 418.241,Z 175.389,A -85,B 0,C 180,E1 -10114.582,E2 -10114.582} C_VEL
LIN {X 0,Y 418.215,Z 175.39,A -85,B 0,C 180,E1 -10117.837,E2 -10117.837} C_VEL
LIN {X 0,Y 418.247,Z 175.386,A -85,B 0,C 180,E1 -10120.945,E2 -10120.945} C_VEL
LIN {X 0,Y 418.249,Z 175.384,A -85,B 0,C 180,E1 -10123.74,E2 -10123.74} C_VEL
LIN {X 0,Y 418.265,Z 175.388,A -85,B 0,C 180,E1 -10126.461,E2 -10126.461} C_VEL
LIN {X 0,Y 418.254,Z 175.4,A -85,B 0,C 180,E1 -10129.694,E2 -10129.694} C_VEL
LIN {X 0,Y 419.147,Z 180.799,A -85,B 0,C 180,E1 -10132.874,E2 -10132.874} C_VEL
LIN {X 0,Y 419.372,Z 184.078,A -85,B 0,C 180,E1 -10134.683,E2 -10134.683} C_VEL
LIN {X 0,Y 418.991,Z 190.624,A -85,B 0,C 180,E1 -10138.108,E2 -10138.108} C_VEL
LIN {X 0,Y 418.519,Z 197.172,A -85,B 0,C 180,E1 -10141.41,E2 -10141.41} C_VEL
LIN {X 0,Y 418.2,Z 203.732,A -85,B 0,C 180,E1 -10144.628,E2 -10144.628} C_VEL
LIN {X 0,Y 417.837,Z 211.341,A -85,B 0,C 180,E1 -10148.284,E2 -10148.284} C_VEL
LIN {X 0,Y 417.498,Z 218.899,A -85,B 0,C 180,E1 -10151.857,E2 -10151.857} C_VEL
LIN {X 0,Y 417.422,Z 221.01,A -85,B 0,C 180,E1 -10152.851,E2 -10152.851} C_VEL
LIN {X 0,Y 419.728,Z 234.393,A -85,B 0,C 180,E1 -10153.343,E2 -10153.343} C_VEL
LIN {X 0,Y 421.398,Z 247.283,A -85,B 0,C 180,E1 -10154.003,E2 -10154.003} C_VEL
LIN {X 0,Y 421.12,Z 255.917,A -85,B 0,C 180,E1 -10154.515,E2 -10154.515} C_VEL
LIN {X 0,Y 420.368,Z 267.268,A -85,B 0,C 180,E1 -10155.354,E2 -10155.354} C_VEL
LIN {X 0,Y 419.608,Z 278.816,A -85,B 0,C 180,E1 -10156.44,E2 -10156.44} C_VEL
LIN {X 0,Y 418.981,Z 289.016,A -85,B 0,C 180,E1 -10157.652,E2 -10157.652} C_VEL
LIN {X 0,Y 418.254,Z 298.827,A -85,B 0,C 180,E1 -10159.105,E2 -10159.105} C_VEL
LIN {X 0,Y 417.762,Z 306.69,A -85,B 0,C 180,E1 -10160.561,E2 -10160.561} C_VEL
LIN {X 0,Y 417.463,Z 312.033,A -85,B 0,C 180,E1 -10161.774,E2 -10161.774} C_VEL
LIN {X 0,Y 417.23,Z 317.244,A -85,B 0,C 180,E1 -10163.23,E2 -10163.23} C_VEL
LIN {X 0,Y 417.123,Z 321.288,A -85,B 0,C 180,E1 -10164.684,E2 -10164.684} C_VEL
LIN {X 0,Y 417.014,Z 324.277,A -85,B 0,C 180,E1 -10166.136,E2 -10166.136} C_VEL
LIN {X 0,Y 417.028,Z 325.73,A -85,B 0,C 180,E1 -10167.103,E2 -10167.103} C_VEL
LIN {X 0,Y 417.056,Z 326.758,A -85,B 0,C 180,E1 -10168.069,E2 -10168.069} C_VEL
LIN {X 0,Y 417.004,Z 327.647,A -85,B 0,C 180,E1 -10170.001,E2 -10170.001} C_VEL
LIN {X 0,Y 417.01,Z 327.484,A -85,B 0,C 180,E1 -10170.966,E2 -10170.966} C_VEL
LIN {X 0,Y 417.056,Z 326.908,A -85,B 0,C 180,E1 -10171.932,E2 -10171.932} C_VEL
LIN {X 0,Y 417.027,Z 325.941,A -85,B 0,C 180,E1 -10172.898,E2 -10172.898} C_VEL
LIN {X 0,Y 417.013,Z 324.581,A -85,B 0,C 180,E1 -10173.866,E2 -10173.866} C_VEL
LIN {X 0,Y 417.121,Z 321.707,A -85,B 0,C 180,E1 -10175.317,E2 -10175.317} C_VEL
LIN {X 0,Y 417.235,Z 317.806,A -85,B 0,C 180,E1 -10176.772,E2 -10176.772} C_VEL
LIN {X 0,Y 417.468,Z 312.78,A -85,B 0,C 180,E1 -10178.227,E2 -10178.227} C_VEL
LIN {X 0,Y 417.865,Z 306.473,A -85,B 0,C 180,E1 -10179.682,E2 -10179.682} C_VEL
LIN {X 0,Y 418.411,Z 298.579,A -85,B 0,C 180,E1 -10181.137,E2 -10181.137} C_VEL
LIN {X 0,Y 419.093,Z 290.545,A -85,B 0,C 180,E1 -10182.346,E2 -10182.346} C_VEL
LIN {X 0,Y 419.737,Z 280.749,A -85,B 0,C 180,E1 -10183.557,E2 -10183.557} C_VEL
LIN {X 0,Y 420.532,Z 269.837,A -85,B 0,C 180,E1 -10184.641,E2 -10184.641} C_VEL
LIN {X 0,Y 421.276,Z 259.152,A -85,B 0,C 180,E1 -10185.481,E2 -10185.481} C_VEL
LIN {X 0,Y 421.868,Z 248.549,A -85,B 0,C 180,E1 -10186.14,E2 -10186.14} C_VEL
LIN {X 0,Y 420.301,Z 235.905,A -85,B 0,C 180,E1 -10186.816,E2 -10186.816} C_VEL
LIN {X 0,Y 417.757,Z 222.703,A -85,B 0,C 180,E1 -10187.358,E2 -10187.358} C_VEL
LIN {X 0,Y 417.462,Z 220.908,A -85,B 0,C 180,E1 -10187.423,E2 -10187.423} C_VEL
LIN {X 0,Y 417.752,Z 214.025,A -85,B 0,C 180,E1 -10190.688,E2 -10190.688} C_VEL
LIN {X 0,Y 418.046,Z 207.617,A -85,B 0,C 180,E1 -10193.795,E2 -10193.795} C_VEL
LIN {X 0,Y 418.446,Z 200.873,A -85,B 0,C 180,E1 -10197.107,E2 -10197.107} C_VEL
LIN {X 0,Y 418.891,Z 194.679,A -85,B 0,C 180,E1 -10200.219,E2 -10200.219} C_VEL
LIN {X 0,Y 419.306,Z 188.24,A -85,B 0,C 180,E1 -10203.579,E2 -10203.579} C_VEL
LIN {X 0,Y 419.47,Z 183.985,A -85,B 0,C 180,E1 -10205.9,E2 -10205.9} C_VEL
LIN {X 0,Y 418.996,Z 179.743,A -85,B 0,C 180,E1 -10208.359,E2 -10208.359} C_VEL
LIN {X 0,Y 418.276,Z 175.383,A -85,B 0,C 180,E1 -10211.098,E2 -10211.098} C_VEL
LIN {X 0,Y 418.273,Z 175.386,A -85,B 0,C 180,E1 -10213.738,E2 -10213.738} C_VEL
LIN {X 0,Y 418.196,Z 175.395,A -85,B 0,C 180,E1 -10216.447,E2 -10216.447} C_VEL
LIN {X 0,Y 418.209,Z 175.392,A -85,B 0,C 180,E1 -10219.129,E2 -10219.129} C_VEL
LIN {X 0,Y 418.209,Z 175.389,A -85,B 0,C 180,E1 -10222.166,E2 -10222.166} C_VEL
LIN {X 0,Y 418.249,Z 175.389,A -85,B 0,C 180,E1 -10225.418,E2 -10225.418} C_VEL
LIN {X 0,Y 418.192,Z 175.392,A -85,B 0,C 180,E1 -10228.602,E2 -10228.602} C_VEL
LIN {X 0,Y 418.271,Z 175.382,A -85,B 0,C 180,E1 -10231.935,E2 -10231.935} C_VEL
LIN {X 0,Y 418.27,Z 175.387,A -85,B 0,C 180,E1 -10235.161,E2 -10235.161} C_VEL
LIN {X 0,Y 418.241,Z 175.385,A -85,B 0,C 180,E1 -10238.304,E2 -10238.304} C_VEL
LIN {X 0,Y 418.264,Z 175.384,A -85,B 0,C 180,E1 -10241.382,E2 -10241.382} C_VEL
LIN {X 0,Y 418.286,Z 175.383,A -85,B 0,C 180,E1 -10244.405,E2 -10244.405} C_VEL
LIN {X 0,Y 418.346,Z 175.372,A -85,B 0,C 180,E1 -10247.385,E2 -10247.385} C_VEL
LIN {X 0,Y 418.34,Z 175.376,A -85,B 0,C 180,E1 -10250.329,E2 -10250.329} C_VEL
LIN {X 0,Y 418.495,Z 175.353,A -85,B 0,C 180,E1 -10253.249,E2 -10253.249} C_VEL
LIN {X 0,Y 418.324,Z 175.375,A -85,B 0,C 180,E1 -10255.182,E2 -10255.182} C_VEL
LIN {X 0,Y 418.514,Z 175.355,A -85,B 0,C 180,E1 -10258.076,E2 -10258.076} C_VEL
LIN {X 0,Y 418.641,Z 175.338,A -85,B 0,C 180,E1 -10260,E2 -10260} C_VEL
LIN {X 0,Y 418.496,Z 175.353,A -85,B 0,C 180,E1 -10262.888,E2 -10262.888} C_VEL
LIN {X 0,Y 418.468,Z 175.357,A -85,B 0,C 180,E1 -10266.604,E2 -10266.604} C_VEL
LIN {X 0,Y 418.316,Z 175.38,A -85,B 0,C 180,E1 -10269.672,E2 -10269.672} C_VEL
LIN {X 0,Y 418.322,Z 175.375,A -85,B 0,C 180,E1 -10273.001,E2 -10273.001} C_VEL
LIN {X 0,Y 418.312,Z 175.375,A -85,B 0,C 180,E1 -10276.746,E2 -10276.746} C_VEL
LIN {X 0,Y 418.249,Z 175.387,A -85,B 0,C 180,E1 -10279.791,E2 -10279.791} C_VEL
LIN {X 0,Y 418.218,Z 175.389,A -85,B 0,C 180,E1 -10282.738,E2 -10282.738} C_VEL
LIN {X 0,Y 418.251,Z 175.385,A -85,B 0,C 180,E1 -10285.906,E2 -10285.906} C_VEL
LIN {X 0,Y 418.256,Z 175.387,A -85,B 0,C 180,E1 -10289.163,E2 -10289.163} C_VEL
LIN {X 0,Y 418.241,Z 175.389,A -85,B 0,C 180,E1 -10292.846,E2 -10292.846} C_VEL
LIN {X 0,Y 418.23,Z 175.387,A -85,B 0,C 180,E1 -10296.24,E2 -10296.24} C_VEL
LIN {X 0,Y 418.232,Z 175.386,A -85,B 0,C 180,E1 -10299.685,E2 -10299.685} C_VEL
LIN {X 0,Y 418.218,Z 175.389,A -85,B 0,C 180,E1 -10302.323,E2 -10302.323} C_VEL
LIN {X 0,Y 418.226,Z 175.389,A -85,B 0,C 180,E1 -10305.111,E2 -10305.111} C_VEL
LIN {X 0,Y 418.231,Z 175.387,A -85,B 0,C 180,E1 -10307.769,E2 -10307.769} C_VEL
LIN {X 0,Y 418.197,Z 175.395,A -85,B 0,C 180,E1 -10310.63,E2 -10310.63} C_VEL
LIN {X 0,Y 418.151,Z 175.693,A -85,B 0,C 180,E1 -10312.181,E2 -10312.181} C_VEL
LIN {X 0,Y 418.13,Z 179.325,A -85,B 0,C 180,E1 -10315.149,E2 -10315.149} C_VEL
LIN {X 0,Y 418.033,Z 182.23,A -85,B 0,C 180,E1 -10317.455,E2 -10317.455} C_VEL
LIN {X 0,Y 417.804,Z 186.843,A -85,B 0,C 180,E1 -10321.011,E2 -10321.011} C_VEL
LIN {X 0,Y 417.634,Z 190.929,A -85,B 0,C 180,E1 -10324.055,E2 -10324.055} C_VEL
LIN {X 0,Y 417.546,Z 193.855,A -85,B 0,C 180,E1 -10326.175,E2 -10326.175} C_VEL
LIN {X 0,Y 417.392,Z 198.248,A -85,B 0,C 180,E1 -10329.293,E2 -10329.293} C_VEL
LIN {X 0,Y 417.418,Z 200.179,A -85,B 0,C 180,E1 -10330.655,E2 -10330.655} C_VEL
LIN {X 0,Y 420.656,Z 214.027,A -85,B 0,C 180,E1 -10331.262,E2 -10331.262} C_VEL
LIN {X 0,Y 422.401,Z 224.193,A -85,B 0,C 180,E1 -10331.823,E2 -10331.823} C_VEL
LIN {X 0,Y 421.799,Z 236.085,A -85,B 0,C 180,E1 -10332.548,E2 -10332.548} C_VEL
LIN {X 0,Y 421.075,Z 246.869,A -85,B 0,C 180,E1 -10333.392,E2 -10333.392} C_VEL
LIN {X 0,Y 420.299,Z 257.847,A -85,B 0,C 180,E1 -10334.482,E2 -10334.482} C_VEL
LIN {X 0,Y 419.545,Z 267.648,A -85,B 0,C 180,E1 -10335.695,E2 -10335.695} C_VEL
LIN {X 0,Y 418.817,Z 276.943,A -85,B 0,C 180,E1 -10337.122,E2 -10337.122} C_VEL
LIN {X 0,Y 418.281,Z 284.648,A -85,B 0,C 180,E1 -10338.614,E2 -10338.614} C_VEL
LIN {X 0,Y 417.719,Z 291.595,A -85,B 0,C 180,E1 -10340.314,E2 -10340.314} C_VEL
LIN {X 0,Y 417.467,Z 296.184,A -85,B 0,C 180,E1 -10341.773,E2 -10341.773} C_VEL
LIN {X 0,Y 417.251,Z 299.674,A -85,B 0,C 180,E1 -10343.229,E2 -10343.229} C_VEL
LIN {X 0,Y 417.152,Z 301.439,A -85,B 0,C 180,E1 -10344.198,E2 -10344.198} C_VEL
LIN {X 0,Y 417.11,Z 302.77,A -85,B 0,C 180,E1 -10345.167,E2 -10345.167} C_VEL
LIN {X 0,Y 417.07,Z 304.269,A -85,B 0,C 180,E1 -10347.102,E2 -10347.102} C_VEL
LIN {X 0,Y 417.074,Z 304.408,A -85,B 0,C 180,E1 -10348.068,E2 -10348.068} C_VEL
LIN {X 0,Y 417.009,Z 303.509,A -85,B 0,C 180,E1 -10349.999,E2 -10349.999} C_VEL
LIN {X 0,Y 417.046,Z 302.487,A -85,B 0,C 180,E1 -10350.965,E2 -10350.965} C_VEL
LIN {X 0,Y 417.217,Z 299.956,A -85,B 0,C 180,E1 -10352.482,E2 -10352.482} C_VEL
LIN {X 0,Y 417.446,Z 296.839,A -85,B 0,C 180,E1 -10353.86,E2 -10353.86} C_VEL
LIN {X 0,Y 417.604,Z 292.473,A -85,B 0,C 180,E1 -10355.31,E2 -10355.31} C_VEL
LIN {X 0,Y 417.868,Z 288.549,A -85,B 0,C 180,E1 -10356.365,E2 -10356.365} C_VEL
LIN {X 0,Y 417.402,Z 285.648,A -85,B 0,C 180,E1 -10357.064,E2 -10357.064} C_VEL
LIN {X 0,Y 413.8,Z 278.44,A -85,B 0,C 180,E1 -10358.625,E2 -10358.625} C_VEL
LIN {X 0,Y 412.243,Z 273.741,A -85,B 0,C 180,E1 -10359.481,E2 -10359.481} C_VEL
LIN {X 0,Y 412.14,Z 271.122,A -85,B 0,C 180,E1 -10359.894,E2 -10359.894} C_VEL
LIN {X 0,Y 412.826,Z 262.746,A -85,B 0,C 180,E1 -10361.04,E2 -10361.04} C_VEL
LIN {X 0,Y 413.5,Z 252.992,A -85,B 0,C 180,E1 -10362.14,E2 -10362.14} C_VEL
LIN {X 0,Y 413.929,Z 245.13,A -85,B 0,C 180,E1 -10362.875,E2 -10362.875} C_VEL
LIN {X 0,Y 414.575,Z 233.976,A -85,B 0,C 180,E1 -10363.727,E2 -10363.727} C_VEL
LIN {X 0,Y 415.138,Z 224.178,A -85,B 0,C 180,E1 -10364.311,E2 -10364.311} C_VEL
LIN {X 0,Y 412.828,Z 211.717,A -85,B 0,C 180,E1 -10364.989,E2 -10364.989} C_VEL
LIN {X 0,Y 410.34,Z 200.341,A -85,B 0,C 180,E1 -10365.457,E2 -10365.457} C_VEL
LIN {X 0,Y 410.425,Z 195.356,A -85,B 0,C 180,E1 -10368.985,E2 -10368.985} C_VEL
LIN {X 0,Y 410.586,Z 190.571,A -85,B 0,C 180,E1 -10372.433,E2 -10372.433} C_VEL
LIN {X 0,Y 410.69,Z 186.734,A -85,B 0,C 180,E1 -10375.326,E2 -10375.326} C_VEL
LIN {X 0,Y 410.865,Z 182.479,A -85,B 0,C 180,E1 -10378.614,E2 -10378.614} C_VEL
LIN {X 0,Y 411.033,Z 178.179,A -85,B 0,C 180,E1 -10382.005,E2 -10382.005} C_VEL
LIN {X 0,Y 411.035,Z 176.749,A -85,B 0,C 180,E1 -10383.168,E2 -10383.168} C_VEL
LIN {X 0,Y 411.13,Z 176.274,A -85,B 0,C 180,E1 -10384.861,E2 -10384.861} C_VEL
LIN {X 0,Y 411.187,Z 176.265,A -85,B 0,C 180,E1 -10388.164,E2 -10388.164} C_VEL
LIN {X 0,Y 411.151,Z 176.272,A -85,B 0,C 180,E1 -10391.225,E2 -10391.225} C_VEL
LIN {X 0,Y 411.172,Z 176.266,A -85,B 0,C 180,E1 -10394.486,E2 -10394.486} C_VEL
LIN {X 0,Y 411.211,Z 176.265,A -85,B 0,C 180,E1 -10397.294,E2 -10397.294} C_VEL
LIN {X 0,Y 411.209,Z 176.264,A -85,B 0,C 180,E1 -10400.774,E2 -10400.774} C_VEL
LIN {X 0,Y 411.175,Z 176.268,A -85,B 0,C 180,E1 -10404.468,E2 -10404.468} C_VEL
LIN {X 0,Y 411.184,Z 176.268,A -85,B 0,C 180,E1 -10406.871,E2 -10406.871} C_VEL
LIN {X 0,Y 411.215,Z 176.264,A -85,B 0,C 180,E1 -10410.64,E2 -10410.64} C_VEL
LIN {X 0,Y 411.213,Z 176.26,A -85,B 0,C 180,E1 -10413.617,E2 -10413.617} C_VEL
LIN {X 0,Y 411.229,Z 176.258,A -85,B 0,C 180,E1 -10417.338,E2 -10417.338} C_VEL
LIN {X 0,Y 411.236,Z 176.26,A -85,B 0,C 180,E1 -10420.029,E2 -10420.029} C_VEL
LIN {X 0,Y 411.233,Z 176.259,A -85,B 0,C 180,E1 -10423.129,E2 -10423.129} C_VEL
LIN {X 0,Y 411.245,Z 176.26,A -85,B 0,C 180,E1 -10426.157,E2 -10426.157} C_VEL
LIN {X 0,Y 411.291,Z 176.251,A -85,B 0,C 180,E1 -10429.166,E2 -10429.166} C_VEL
LIN {X 0,Y 411.449,Z 176.235,A -85,B 0,C 180,E1 -10432.146,E2 -10432.146} C_VEL
LIN {X 0,Y 411.472,Z 176.232,A -85,B 0,C 180,E1 -10434.118,E2 -10434.118} C_VEL
LIN {X 0,Y 411.477,Z 176.231,A -85,B 0,C 180,E1 -10438.042,E2 -10438.042} C_VEL
LIN {X 0,Y 411.604,Z 176.215,A -85,B 0,C 180,E1 -10440,E2 -10440} C_VEL
LIN {X 0,Y 411.443,Z 176.233,A -85,B 0,C 180,E1 -10442.937,E2 -10442.937} C_VEL
LIN {X 0,Y 411.464,Z 176.233,A -85,B 0,C 180,E1 -10445.882,E2 -10445.882} C_VEL
LIN {X 0,Y 411.348,Z 176.244,A -85,B 0,C 180,E1 -10448.845,E2 -10448.845} C_VEL
